LIN {X 0,Y 320.282,Z 387.307,A -85,B 0,C 180,E1 -15901.85,E2 -15901.85} C_VEL
LIN {X 0,Y 317.644,Z 401.035,A -85,B 0,C 180,E1 -15903.382,E2 -15903.382} C_VEL
LIN {X 0,Y 315.007,Z 413.467,A -85,B 0,C 180,E1 -15905.095,E2 -15905.095} C_VEL
LIN {X 0,Y 312.778,Z 423.901,A -85,B 0,C 180,E1 -15906.846,E2 -15906.846} C_VEL
LIN {X 0,Y 310.716,Z 433.586,A -85,B 0,C 180,E1 -15908.783,E2 -15908.783} C_VEL
LIN {X 0,Y 308.469,Z 443.101,A -85,B 0,C 180,E1 -15911.055,E2 -15911.055} C_VEL
LIN {X 0,Y 306.764,Z 451.036,A -85,B 0,C 180,E1 -15913.359,E2 -15913.359} C_VEL
LIN {X 0,Y 305.36,Z 458.451,A -85,B 0,C 180,E1 -15916.015,E2 -15916.015} C_VEL
LIN {X 0,Y 304.367,Z 464.336,A -85,B 0,C 180,E1 -15918.681,E2 -15918.681} C_VEL
LIN {X 0,Y 303.943,Z 467.84,A -85,B 0,C 180,E1 -15920.685,E2 -15920.685} C_VEL
LIN {X 0,Y 303.628,Z 471.382,A -85,B 0,C 180,E1 -15923.354,E2 -15923.354} C_VEL
LIN {X 0,Y 303.568,Z 473.714,A -85,B 0,C 180,E1 -15926.017,E2 -15926.017} C_VEL
LIN {X 0,Y 303.569,Z 474.886,A -85,B 0,C 180,E1 -15928.673,E2 -15928.673} C_VEL
LIN {X 0,Y 303.569,Z 474.883,A -85,B 0,C 180,E1 -15931.327,E2 -15931.327} C_VEL
LIN {X 0,Y 303.568,Z 473.697,A -85,B 0,C 180,E1 -15933.983,E2 -15933.983} C_VEL
LIN {X 0,Y 303.628,Z 471.354,A -85,B 0,C 180,E1 -15936.646,E2 -15936.646} C_VEL
LIN {X 0,Y 303.943,Z 467.807,A -85,B 0,C 180,E1 -15939.315,E2 -15939.315} C_VEL
LIN {X 0,Y 304.596,Z 462.968,A -85,B 0,C 180,E1 -15941.985,E2 -15941.985} C_VEL
LIN {X 0,Y 305.622,Z 456.707,A -85,B 0,C 180,E1 -15944.652,E2 -15944.652} C_VEL
LIN {X 0,Y 307.21,Z 448.855,A -85,B 0,C 180,E1 -15947.301,E2 -15947.301} C_VEL
LIN {X 0,Y 308.97,Z 440.507,A -85,B 0,C 180,E1 -15949.604,E2 -15949.604} C_VEL
LIN {X 0,Y 311.289,Z 430.696,A -85,B 0,C 180,E1 -15951.821,E2 -15951.821} C_VEL
LIN {X 0,Y 313.52,Z 420.19,A -85,B 0,C 180,E1 -15953.797,E2 -15953.797} C_VEL
LIN {X 0,Y 316.153,Z 407.953,A -85,B 0,C 180,E1 -15955.689,E2 -15955.689} C_VEL
LIN {X 0,Y 318.912,Z 394.331,A -85,B 0,C 180,E1 -15957.389,E2 -15957.389} C_VEL
LIN {X 0,Y 321.417,Z 380.677,A -85,B 0,C 180,E1 -15958.754,E2 -15958.754} C_VEL
LIN {X 0,Y 323.433,Z 367.3,A -85,B 0,C 180,E1 -15959.83,E2 -15959.83} C_VEL
LIN {X 0,Y 325.217,Z 353.283,A -85,B 0,C 180,E1 -15960.7,E2 -15960.7} C_VEL
LIN {X 0,Y 326.763,Z 337.925,A -85,B 0,C 180,E1 -15961.392,E2 -15961.392} C_VEL
LIN {X 0,Y 327.693,Z 323.115,A -85,B 0,C 180,E1 -15961.834,E2 -15961.834} C_VEL
LIN {X 0,Y 330.786,Z 234.22,A -85,B 0,C 180,E1 -15963.753,E2 -15963.753} C_VEL
LIN {X 0,Y 331.307,Z 215.247,A -85,B 0,C 180,E1 -15964.177,E2 -15964.177} C_VEL
LIN {X 0,Y 328.979,Z 201.739,A -85,B 0,C 180,E1 -15964.801,E2 -15964.801} C_VEL
LIN {X 0,Y 319.968,Z 182.03,A -85,B 0,C 180,E1 -15966.456,E2 -15966.456} C_VEL
LIN {X 0,Y 313.395,Z 169.255,A -85,B 0,C 180,E1 -15967.703,E2 -15967.703} C_VEL
LIN {X 0,Y 309.541,Z 161.949,A -85,B 0,C 180,E1 -15968.469,E2 -15968.469} C_VEL
LIN {X 0,Y 306.572,Z 151.906,A -85,B 0,C 180,E1 -15971.668,E2 -15971.668} C_VEL
LIN {X 0,Y 305.43,Z 148.062,A -85,B 0,C 180,E1 -15972.974,E2 -15972.974} C_VEL
LIN {X 0,Y 305.455,Z 148.059,A -85,B 0,C 180,E1 -15977.414,E2 -15977.414} C_VEL
LIN {X 0,Y 305.468,Z 148.053,A -85,B 0,C 180,E1 -15981.597,E2 -15981.597} C_VEL
LIN {X 0,Y 305.463,Z 148.054,A -85,B 0,C 180,E1 -15984.887,E2 -15984.887} C_VEL
LIN {X 0,Y 305.453,Z 148.058,A -85,B 0,C 180,E1 -15988.355,E2 -15988.355} C_VEL
LIN {X 0,Y 305.522,Z 148.05,A -85,B 0,C 180,E1 -15991.114,E2 -15991.114} C_VEL
LIN {X 0,Y 305.573,Z 148.045,A -85,B 0,C 180,E1 -15994.088,E2 -15994.088} C_VEL
LIN {X 0,Y 305.502,Z 148.056,A -85,B 0,C 180,E1 -15998.403,E2 -15998.403} C_VEL
LIN {X 0,Y 305.592,Z 148.044,A -85,B 0,C 180,E1 -16001.218,E2 -16001.218} C_VEL
LIN {X 0,Y 305.651,Z 148.037,A -85,B 0,C 180,E1 -16005.349,E2 -16005.349} C_VEL
LIN {X 0,Y 305.626,Z 148.04,A -85,B 0,C 180,E1 -16009.399,E2 -16009.399} C_VEL
LIN {X 0,Y 305.748,Z 148.015,A -85,B 0,C 180,E1 -16012.073,E2 -16012.073} C_VEL
LIN {X 0,Y 305.668,Z 148.031,A -85,B 0,C 180,E1 -16014.723,E2 -16014.723} C_VEL
LIN {X 0,Y 305.942,Z 147.999,A -85,B 0,C 180,E1 -16018.684,E2 -16018.684} C_VEL
LIN {X 0,Y 305.949,Z 147.996,A -85,B 0,C 180,E1 -16021.316,E2 -16021.316} C_VEL
LIN {X 0,Y 305.789,Z 148.021,A -85,B 0,C 180,E1 -16026.599,E2 -16026.599} C_VEL
LIN {X 0,Y 305.696,Z 148.022,A -85,B 0,C 180,E1 -16029.261,E2 -16029.261} C_VEL
LIN {X 0,Y 305.573,Z 148.037,A -85,B 0,C 180,E1 -16033.297,E2 -16033.297} C_VEL
LIN {X 0,Y 305.533,Z 148.043,A -85,B 0,C 180,E1 -16037.4,E2 -16037.4} C_VEL
LIN {X 0,Y 305.501,Z 148.051,A -85,B 0,C 180,E1 -16040.186,E2 -16040.186} C_VEL
LIN {X 0,Y 305.475,Z 148.051,A -85,B 0,C 180,E1 -16044.464,E2 -16044.464} C_VEL
LIN {X 0,Y 305.455,Z 148.035,A -85,B 0,C 180,E1 -16047.398,E2 -16047.398} C_VEL
LIN {X 0,Y 305.431,Z 148.063,A -85,B 0,C 180,E1 -16050.413,E2 -16050.413} C_VEL
LIN {X 0,Y 305.466,Z 148.053,A -85,B 0,C 180,E1 -16054.078,E2 -16054.078} C_VEL
LIN {X 0,Y 305.455,Z 148.057,A -85,B 0,C 180,E1 -16056.742,E2 -16056.742} C_VEL
LIN {X 0,Y 305.41,Z 148.062,A -85,B 0,C 180,E1 -16060.59,E2 -16060.59} C_VEL
LIN {X 0,Y 305.421,Z 148.064,A -85,B 0,C 180,E1 -16063.656,E2 -16063.656} C_VEL
LIN {X 0,Y 305.436,Z 148.064,A -85,B 0,C 180,E1 -16067.418,E2 -16067.418} C_VEL
LIN {X 0,Y 305.445,Z 148.217,A -85,B 0,C 180,E1 -16070.766,E2 -16070.766} C_VEL
LIN {X 0,Y 305.708,Z 149.306,A -85,B 0,C 180,E1 -16071.033,E2 -16071.033} C_VEL
LIN {X 0,Y 307.015,Z 151.728,A -85,B 0,C 180,E1 -16071.303,E2 -16071.303} C_VEL
LIN {X 0,Y 311.31,Z 158.512,A -85,B 0,C 180,E1 -16072.134,E2 -16072.134} C_VEL
LIN {X 0,Y 319.576,Z 173.575,A -85,B 0,C 180,E1 -16073.7,E2 -16073.7} C_VEL
LIN {X 0,Y 326.924,Z 188.491,A -85,B 0,C 180,E1 -16075.041,E2 -16075.041} C_VEL
LIN {X 0,Y 331.801,Z 199.525,A -85,B 0,C 180,E1 -16075.917,E2 -16075.917} C_VEL
LIN {X 0,Y 330.462,Z 240.875,A -85,B 0,C 180,E1 -16076.819,E2 -16076.819} C_VEL
LIN {X 0,Y 327.848,Z 313.454,A -85,B 0,C 180,E1 -16078.408,E2 -16078.408} C_VEL
LIN {X 0,Y 326.848,Z 327.773,A -85,B 0,C 180,E1 -16078.932,E2 -16078.932} C_VEL
LIN {X 0,Y 325.558,Z 340.971,A -85,B 0,C 180,E1 -16079.614,E2 -16079.614} C_VEL
LIN {X 0,Y 323.859,Z 355.279,A -85,B 0,C 180,E1 -16080.595,E2 -16080.595} C_VEL
LIN {X 0,Y 321.646,Z 369.25,A -85,B 0,C 180,E1 -16081.803,E2 -16081.803} C_VEL
LIN {X 0,Y 319.391,Z 382.018,A -85,B 0,C 180,E1 -16083.186,E2 -16083.186} C_VEL
LIN {X 0,Y 316.811,Z 394.879,A -85,B 0,C 180,E1 -16084.896,E2 -16084.896} C_VEL
LIN {X 0,Y 314.858,Z 403.853,A -85,B 0,C 180,E1 -16086.31,E2 -16086.31} C_VEL
LIN {X 0,Y 312.98,Z 412.416,A -85,B 0,C 180,E1 -16087.906,E2 -16087.906} C_VEL
LIN {X 0,Y 310.65,Z 422.648,A -85,B 0,C 180,E1 -16090.162,E2 -16090.162} C_VEL
LIN {X 0,Y 308.592,Z 431.143,A -85,B 0,C 180,E1 -16092.437,E2 -16092.437} C_VEL
LIN {X 0,Y 307.076,Z 438.205,A -85,B 0,C 180,E1 -16094.74,E2 -16094.74} C_VEL
LIN {X 0,Y 305.643,Z 444.756,A -85,B 0,C 180,E1 -16097.382,E2 -16097.382} C_VEL
LIN {X 0,Y 304.74,Z 449.87,A -85,B 0,C 180,E1 -16100.04,E2 -16100.04} C_VEL
LIN {X 0,Y 304.281,Z 452.816,A -85,B 0,C 180,E1 -16102.034,E2 -16102.034} C_VEL
LIN {X 0,Y 303.871,Z 455.7,A -85,B 0,C 180,E1 -16104.692,E2 -16104.692} C_VEL
LIN {X 0,Y 303.673,Z 457.433,A -85,B 0,C 180,E1 -16107.347,E2 -16107.347} C_VEL
LIN {X 0,Y 303.609,Z 458.038,A -85,B 0,C 180,E1 -16110,E2 -16110} C_VEL
LIN {X 0,Y 303.672,Z 457.475,A -85,B 0,C 180,E1 -16112.653,E2 -16112.653} C_VEL
LIN {X 0,Y 303.87,Z 455.798,A -85,B 0,C 180,E1 -16115.308,E2 -16115.308} C_VEL
LIN {X 0,Y 304.274,Z 452.967,A -85,B 0,C 180,E1 -16117.966,E2 -16117.966} C_VEL
LIN {X 0,Y 304.917,Z 448.913,A -85,B 0,C 180,E1 -16120.626,E2 -16120.626} C_VEL
LIN {X 0,Y 305.957,Z 443.534,A -85,B 0,C 180,E1 -16123.28,E2 -16123.28} C_VEL
LIN {X 0,Y 307.039,Z 438.509,A -85,B 0,C 180,E1 -16125.262,E2 -16125.262} C_VEL
LIN {X 0,Y 308.808,Z 430.409,A -85,B 0,C 180,E1 -16127.893,E2 -16127.893} C_VEL
LIN {X 0,Y 310.834,Z 421.751,A -85,B 0,C 180,E1 -16130.17,E2 -16130.17} C_VEL
LIN {X 0,Y 313.314,Z 411.331,A -85,B 0,C 180,E1 -16132.416,E2 -16132.416} C_VEL
LIN {X 0,Y 315.625,Z 400.631,A -85,B 0,C 180,E1 -16134.326,E2 -16134.326} C_VEL
LIN {X 0,Y 317.873,Z 390.102,A -85,B 0,C 180,E1 -16135.891,E2 -16135.891} C_VEL
LIN {X 0,Y 320.214,Z 377.582,A -85,B 0,C 180,E1 -16137.446,E2 -16137.446} C_VEL
LIN {X 0,Y 322.645,Z 363.942,A -85,B 0,C 180,E1 -16138.799,E2 -16138.799} C_VEL
LIN {X 0,Y 324.486,Z 350.567,A -85,B 0,C 180,E1 -16139.878,E2 -16139.878} C_VEL
LIN {X 0,Y 326.118,Z 335.98,A -85,B 0,C 180,E1 -16140.785,E2 -16140.785} C_VEL
LIN {X 0,Y 327.451,Z 320.953,A -85,B 0,C 180,E1 -16141.454,E2 -16141.454} C_VEL
LIN {X 0,Y 328.374,Z 305.322,A -85,B 0,C 180,E1 -16141.896,E2 -16141.896} C_VEL
LIN {X 0,Y 331.426,Z 216.152,A -85,B 0,C 180,E1 -16143.819,E2 -16143.819} C_VEL
LIN {X 0,Y 331.182,Z 212.313,A -85,B 0,C 180,E1 -16143.946,E2 -16143.946} C_VEL
LIN {X 0,Y 329.668,Z 206.897,A -85,B 0,C 180,E1 -16144.265,E2 -16144.265} C_VEL
LIN {X 0,Y 327.311,Z 201.936,A -85,B 0,C 180,E1 -16144.678,E2 -16144.678} C_VEL
LIN {X 0,Y 321.759,Z 192.218,A -85,B 0,C 180,E1 -16145.631,E2 -16145.631} C_VEL
LIN {X 0,Y 320.189,Z 188.776,A -85,B 0,C 180,E1 -16145.927,E2 -16145.927} C_VEL
LIN {X 0,Y 311.448,Z 171.517,A -85,B 0,C 180,E1 -16147.6,E2 -16147.6} C_VEL
LIN {X 0,Y 304.534,Z 159.472,A -85,B 0,C 180,E1 -16148.973,E2 -16148.973} C_VEL
LIN {X 0,Y 300.514,Z 153.176,A -85,B 0,C 180,E1 -16149.792,E2 -16149.792} C_VEL
LIN {X 0,Y 298.852,Z 150.776,A -85,B 0,C 180,E1 -16150.134,E2 -16150.134} C_VEL
LIN {X 0,Y 298.381,Z 148.995,A -85,B 0,C 180,E1 -16150.317,E2 -16150.317} C_VEL
LIN {X 0,Y 298.371,Z 148.945,A -85,B 0,C 180,E1 -16153.097,E2 -16153.097} C_VEL
LIN {X 0,Y 298.37,Z 148.928,A -85,B 0,C 180,E1 -16156.915,E2 -16156.915} C_VEL
LIN {X 0,Y 298.357,Z 148.938,A -85,B 0,C 180,E1 -16161.018,E2 -16161.018} C_VEL
LIN {X 0,Y 298.405,Z 148.924,A -85,B 0,C 180,E1 -16163.928,E2 -16163.928} C_VEL
LIN {X 0,Y 298.393,Z 148.925,A -85,B 0,C 180,E1 -16167.199,E2 -16167.199} C_VEL
LIN {X 0,Y 298.405,Z 148.939,A -85,B 0,C 180,E1 -16171.898,E2 -16171.898} C_VEL
LIN {X 0,Y 298.422,Z 148.935,A -85,B 0,C 180,E1 -16174.918,E2 -16174.918} C_VEL
LIN {X 0,Y 298.417,Z 148.937,A -85,B 0,C 180,E1 -16179.313,E2 -16179.313} C_VEL
LIN {X 0,Y 298.452,Z 148.925,A -85,B 0,C 180,E1 -16182.174,E2 -16182.174} C_VEL
LIN {X 0,Y 298.588,Z 148.914,A -85,B 0,C 180,E1 -16184.994,E2 -16184.994} C_VEL
LIN {X 0,Y 298.586,Z 148.916,A -85,B 0,C 180,E1 -16189.146,E2 -16189.146} C_VEL
LIN {X 0,Y 298.699,Z 148.896,A -85,B 0,C 180,E1 -16191.884,E2 -16191.884} C_VEL
LIN {X 0,Y 298.629,Z 148.904,A -85,B 0,C 180,E1 -16194.598,E2 -16194.598} C_VEL
LIN {X 0,Y 298.914,Z 148.873,A -85,B 0,C 180,E1 -16198.653,E2 -16198.653} C_VEL
LIN {X 0,Y 298.911,Z 148.871,A -85,B 0,C 180,E1 -16201.347,E2 -16201.347} C_VEL
LIN {X 0,Y 298.637,Z 148.901,A -85,B 0,C 180,E1 -16205.401,E2 -16205.401} C_VEL
LIN {X 0,Y 298.71,Z 148.894,A -85,B 0,C 180,E1 -16208.82,E2 -16208.82} C_VEL
LIN {X 0,Y 298.553,Z 148.921,A -85,B 0,C 180,E1 -16212.231,E2 -16212.231} C_VEL
LIN {X 0,Y 298.55,Z 148.92,A -85,B 0,C 180,E1 -16215.168,E2 -16215.168} C_VEL
LIN {X 0,Y 298.51,Z 148.923,A -85,B 0,C 180,E1 -16219.245,E2 -16219.245} C_VEL
LIN {X 0,Y 298.426,Z 148.937,A -85,B 0,C 180,E1 -16223.6,E2 -16223.6} C_VEL
LIN {X 0,Y 298.418,Z 148.93,A -85,B 0,C 180,E1 -16226.581,E2 -16226.581} C_VEL
LIN {X 0,Y 298.402,Z 148.94,A -85,B 0,C 180,E1 -16229.643,E2 -16229.643} C_VEL
LIN {X 0,Y 298.394,Z 148.936,A -85,B 0,C 180,E1 -16232.8,E2 -16232.8} C_VEL
LIN {X 0,Y 298.447,Z 148.927,A -85,B 0,C 180,E1 -16236.807,E2 -16236.807} C_VEL
LIN {X 0,Y 298.389,Z 148.943,A -85,B 0,C 180,E1 -16241.088,E2 -16241.088} C_VEL
LIN {X 0,Y 298.399,Z 148.938,A -85,B 0,C 180,E1 -16243.103,E2 -16243.103} C_VEL
LIN {X 0,Y 298.387,Z 149.027,A -85,B 0,C 180,E1 -16246.102,E2 -16246.102} C_VEL
LIN {X 0,Y 301.743,Z 159.889,A -85,B 0,C 180,E1 -16249.803,E2 -16249.803} C_VEL
LIN {X 0,Y 302.402,Z 162.037,A -85,B 0,C 180,E1 -16250.425,E2 -16250.425} C_VEL
LIN {X 0,Y 312.165,Z 180.214,A -85,B 0,C 180,E1 -16252.4,E2 -16252.4} C_VEL
LIN {X 0,Y 320.694,Z 198.338,A -85,B 0,C 180,E1 -16254.049,E2 -16254.049} C_VEL
LIN {X 0,Y 323.674,Z 205.479,A -85,B 0,C 180,E1 -16254.618,E2 -16254.618} C_VEL
LIN {X 0,Y 325.588,Z 217.919,A -85,B 0,C 180,E1 -16255.183,E2 -16255.183} C_VEL
LIN {X 0,Y 321.554,Z 326.838,A -85,B 0,C 180,E1 -16257.577,E2 -16257.577} C_VEL
LIN {X 0,Y 320.415,Z 341.93,A -85,B 0,C 180,E1 -16258.097,E2 -16258.097} C_VEL
LIN {X 0,Y 318.626,Z 357.365,A -85,B 0,C 180,E1 -16258.871,E2 -16258.871} C_VEL
LIN {X 0,Y 316.699,Z 371.078,A -85,B 0,C 180,E1 -16259.81,E2 -16259.81} C_VEL
LIN {X 0,Y 314.58,Z 383.941,A -85,B 0,C 180,E1 -16260.927,E2 -16260.927} C_VEL
LIN {X 0,Y 312.061,Z 396.955,A -85,B 0,C 180,E1 -16262.322,E2 -16262.322} C_VEL
LIN {X 0,Y 309.265,Z 410.05,A -85,B 0,C 180,E1 -16264.058,E2 -16264.058} C_VEL
LIN {X 0,Y 306.578,Z 421.907,A -85,B 0,C 180,E1 -16265.989,E2 -16265.989} C_VEL
LIN {X 0,Y 304.366,Z 432.073,A -85,B 0,C 180,E1 -16268.004,E2 -16268.004} C_VEL
LIN {X 0,Y 301.959,Z 441.661,A -85,B 0,C 180,E1 -16270.276,E2 -16270.276} C_VEL
LIN {X 0,Y 300.111,Z 449.82,A -85,B 0,C 180,E1 -16272.628,E2 -16272.628} C_VEL
LIN {X 0,Y 298.712,Z 456.572,A -85,B 0,C 180,E1 -16275.001,E2 -16275.001} C_VEL
LIN {X 0,Y 297.615,Z 462.812,A -85,B 0,C 180,E1 -16277.729,E2 -16277.729} C_VEL
LIN {X 0,Y 296.896,Z 467.641,A -85,B 0,C 180,E1 -16280.462,E2 -16280.462} C_VEL
LIN {X 0,Y 296.548,Z 471.183,A -85,B 0,C 180,E1 -16283.195,E2 -16283.195} C_VEL
LIN {X 0,Y 296.469,Z 473.515,A -85,B 0,C 180,E1 -16285.922,E2 -16285.922} C_VEL
LIN {X 0,Y 296.488,Z 474.688,A -85,B 0,C 180,E1 -16288.642,E2 -16288.642} C_VEL
LIN {X 0,Y 296.488,Z 474.684,A -85,B 0,C 180,E1 -16291.358,E2 -16291.358} C_VEL
LIN {X 0,Y 296.469,Z 473.498,A -85,B 0,C 180,E1 -16294.078,E2 -16294.078} C_VEL
LIN {X 0,Y 296.547,Z 471.154,A -85,B 0,C 180,E1 -16296.805,E2 -16296.805} C_VEL
LIN {X 0,Y 296.895,Z 467.606,A -85,B 0,C 180,E1 -16299.538,E2 -16299.538} C_VEL
LIN {X 0,Y 297.609,Z 462.767,A -85,B 0,C 180,E1 -16302.271,E2 -16302.271} C_VEL
LIN {X 0,Y 298.657,Z 456.504,A -85,B 0,C 180,E1 -16305.002,E2 -16305.002} C_VEL
LIN {X 0,Y 300.353,Z 448.652,A -85,B 0,C 180,E1 -16307.709,E2 -16307.709} C_VEL
LIN {X 0,Y 302.223,Z 440.305,A -85,B 0,C 180,E1 -16310.06,E2 -16310.06} C_VEL
LIN {X 0,Y 304.537,Z 430.85,A -85,B 0,C 180,E1 -16312.248,E2 -16312.248} C_VEL
LIN {X 0,Y 306.991,Z 419.987,A -85,B 0,C 180,E1 -16314.335,E2 -16314.335} C_VEL
LIN {X 0,Y 309.728,Z 407.75,A -85,B 0,C 180,E1 -16316.262,E2 -16316.262} C_VEL
LIN {X 0,Y 312.58,Z 394.127,A -85,B 0,C 180,E1 -16317.992,E2 -16317.992} C_VEL
LIN {X 0,Y 315.185,Z 380.472,A -85,B 0,C 180,E1 -16319.377,E2 -16319.377} C_VEL
LIN {X 0,Y 317.382,Z 366.271,A -85,B 0,C 180,E1 -16320.53,E2 -16320.53} C_VEL
LIN {X 0,Y 319.32,Z 351.754,A -85,B 0,C 180,E1 -16321.423,E2 -16321.423} C_VEL
LIN {X 0,Y 320.806,Z 336.793,A -85,B 0,C 180,E1 -16322.09,E2 -16322.09} C_VEL
LIN {X 0,Y 321.751,Z 321.39,A -85,B 0,C 180,E1 -16322.54,E2 -16322.54} C_VEL
LIN {X 0,Y 324.847,Z 235.601,A -85,B 0,C 180,E1 -16324.414,E2 -16324.414} C_VEL
LIN {X 0,Y 325.425,Z 216.339,A -85,B 0,C 180,E1 -16324.849,E2 -16324.849} C_VEL
LIN {X 0,Y 323.337,Z 204.486,A -85,B 0,C 180,E1 -16325.42,E2 -16325.42} C_VEL
LIN {X 0,Y 314.903,Z 185.886,A -85,B 0,C 180,E1 -16327.027,E2 -16327.027} C_VEL
LIN {X 0,Y 308.532,Z 173.387,A -85,B 0,C 180,E1 -16328.279,E2 -16328.279} C_VEL
LIN {X 0,Y 303.597,Z 164.547,A -85,B 0,C 180,E1 -16329.275,E2 -16329.275} C_VEL
LIN {X 0,Y 302.195,Z 161.662,A -85,B 0,C 180,E1 -16329.591,E2 -16329.591} C_VEL
LIN {X 0,Y 299.183,Z 151.637,A -85,B 0,C 180,E1 -16332.94,E2 -16332.94} C_VEL
LIN {X 0,Y 298.385,Z 148.942,A -85,B 0,C 180,E1 -16333.954,E2 -16333.954} C_VEL
LIN {X 0,Y 298.403,Z 148.935,A -85,B 0,C 180,E1 -16336.921,E2 -16336.921} C_VEL
LIN {X 0,Y 298.399,Z 148.935,A -85,B 0,C 180,E1 -16341.008,E2 -16341.008} C_VEL
LIN {X 0,Y 298.418,Z 148.929,A -85,B 0,C 180,E1 -16343.93,E2 -16343.93} C_VEL
LIN {X 0,Y 298.397,Z 148.938,A -85,B 0,C 180,E1 -16347.983,E2 -16347.983} C_VEL
LIN {X 0,Y 298.465,Z 148.93,A -85,B 0,C 180,E1 -16351.905,E2 -16351.905} C_VEL
LIN {X 0,Y 298.487,Z 148.931,A -85,B 0,C 180,E1 -16354.924,E2 -16354.924} C_VEL
LIN {X 0,Y 298.451,Z 148.927,A -85,B 0,C 180,E1 -16359.316,E2 -16359.316} C_VEL
LIN {X 0,Y 298.54,Z 148.923,A -85,B 0,C 180,E1 -16362.18,E2 -16362.18} C_VEL
LIN {X 0,Y 298.595,Z 148.915,A -85,B 0,C 180,E1 -16364.995,E2 -16364.995} C_VEL
LIN {X 0,Y 298.585,Z 148.918,A -85,B 0,C 180,E1 -16369.146,E2 -16369.146} C_VEL
LIN {X 0,Y 298.7,Z 148.892,A -85,B 0,C 180,E1 -16371.884,E2 -16371.884} C_VEL
LIN {X 0,Y 298.637,Z 148.908,A -85,B 0,C 180,E1 -16374.599,E2 -16374.599} C_VEL
LIN {X 0,Y 298.91,Z 148.875,A -85,B 0,C 180,E1 -16378.653,E2 -16378.653} C_VEL
LIN {X 0,Y 298.915,Z 148.873,A -85,B 0,C 180,E1 -16381.347,E2 -16381.347} C_VEL
LIN {X 0,Y 298.737,Z 148.898,A -85,B 0,C 180,E1 -16386.755,E2 -16386.755} C_VEL
LIN {X 0,Y 298.627,Z 148.903,A -85,B 0,C 180,E1 -16389.482,E2 -16389.482} C_VEL
LIN {X 0,Y 298.525,Z 148.915,A -85,B 0,C 180,E1 -16393.617,E2 -16393.617} C_VEL
LIN {X 0,Y 298.464,Z 148.926,A -85,B 0,C 180,E1 -16396.414,E2 -16396.414} C_VEL
LIN {X 0,Y 298.488,Z 148.93,A -85,B 0,C 180,E1 -16399.641,E2 -16399.641} C_VEL
LIN {X 0,Y 298.422,Z 148.936,A -85,B 0,C 180,E1 -16403.601,E2 -16403.601} C_VEL
LIN {X 0,Y 298.408,Z 148.908,A -85,B 0,C 180,E1 -16406.582,E2 -16406.582} C_VEL
LIN {X 0,Y 298.394,Z 148.943,A -85,B 0,C 180,E1 -16409.644,E2 -16409.644} C_VEL
LIN {X 0,Y 298.394,Z 148.941,A -85,B 0,C 180,E1 -16412.801,E2 -16412.801} C_VEL
LIN {X 0,Y 298.429,Z 148.931,A -85,B 0,C 180,E1 -16416.803,E2 -16416.803} C_VEL
LIN {X 0,Y 298.375,Z 148.937,A -85,B 0,C 180,E1 -16419.492,E2 -16419.492} C_VEL
LIN {X 0,Y 298.371,Z 148.94,A -85,B 0,C 180,E1 -16423.097,E2 -16423.097} C_VEL
LIN {X 0,Y 298.371,Z 148.941,A -85,B 0,C 180,E1 -16426.915,E2 -16426.915} C_VEL
LIN {X 0,Y 298.384,Z 149.054,A -85,B 0,C 180,E1 -16429.835,E2 -16429.835} C_VEL
LIN {X 0,Y 299.497,Z 151.955,A -85,B 0,C 180,E1 -16430.139,E2 -16430.139} C_VEL
LIN {X 0,Y 301.215,Z 154.199,A -85,B 0,C 180,E1 -16430.482,E2 -16430.482} C_VEL
LIN {X 0,Y 308.565,Z 166.283,A -85,B 0,C 180,E1 -16431.959,E2 -16431.959} C_VEL
LIN {X 0,Y 316.644,Z 181.593,A -85,B 0,C 180,E1 -16433.528,E2 -16433.528} C_VEL
LIN {X 0,Y 324.076,Z 197.348,A -85,B 0,C 180,E1 -16434.922,E2 -16434.922} C_VEL
LIN {X 0,Y 325.912,Z 201.621,A -85,B 0,C 180,E1 -16435.262,E2 -16435.262} C_VEL
LIN {X 0,Y 323.491,Z 271.441,A -85,B 0,C 180,E1 -16436.801,E2 -16436.801} C_VEL
LIN {X 0,Y 321.834,Z 313.669,A -85,B 0,C 180,E1 -16437.748,E2 -16437.748} C_VEL
LIN {X 0,Y 320.791,Z 327.984,A -85,B 0,C 180,E1 -16438.278,E2 -16438.278} C_VEL
LIN {X 0,Y 319.385,Z 341.953,A -85,B 0,C 180,E1 -16439.018,E2 -16439.018} C_VEL
LIN {X 0,Y 317.695,Z 355.485,A -85,B 0,C 180,E1 -16439.966,E2 -16439.966} C_VEL
LIN {X 0,Y 315.416,Z 369.454,A -85,B 0,C 180,E1 -16441.194,E2 -16441.194} C_VEL
LIN {X 0,Y 313.071,Z 382.221,A -85,B 0,C 180,E1 -16442.6,E2 -16442.6} C_VEL
LIN {X 0,Y 310.37,Z 395.083,A -85,B 0,C 180,E1 -16444.338,E2 -16444.338} C_VEL
LIN {X 0,Y 308.06,Z 405.449,A -85,B 0,C 180,E1 -16446.036,E2 -16446.036} C_VEL
LIN {X 0,Y 306.021,Z 414.236,A -85,B 0,C 180,E1 -16447.732,E2 -16447.732} C_VEL
LIN {X 0,Y 303.622,Z 424.194,A -85,B 0,C 180,E1 -16450.036,E2 -16450.036} C_VEL
LIN {X 0,Y 301.511,Z 432.453,A -85,B 0,C 180,E1 -16452.361,E2 -16452.361} C_VEL
LIN {X 0,Y 299.83,Z 440.199,A -85,B 0,C 180,E1 -16455.058,E2 -16455.058} C_VEL
LIN {X 0,Y 298.391,Z 446.367,A -85,B 0,C 180,E1 -16457.762,E2 -16457.762} C_VEL
LIN {X 0,Y 297.538,Z 451.123,A -85,B 0,C 180,E1 -16460.483,E2 -16460.483} C_VEL
LIN {X 0,Y 297,Z 454.604,A -85,B 0,C 180,E1 -16463.205,E2 -16463.205} C_VEL
LIN {X 0,Y 296.703,Z 456.905,A -85,B 0,C 180,E1 -16465.925,E2 -16465.925} C_VEL
LIN {X 0,Y 296.526,Z 458.08,A -85,B 0,C 180,E1 -16468.642,E2 -16468.642} C_VEL
LIN {X 0,Y 296.526,Z 458.094,A -85,B 0,C 180,E1 -16471.358,E2 -16471.358} C_VEL
LIN {X 0,Y 296.703,Z 456.975,A -85,B 0,C 180,E1 -16474.075,E2 -16474.075} C_VEL
LIN {X 0,Y 296.999,Z 454.729,A -85,B 0,C 180,E1 -16476.795,E2 -16476.795} C_VEL
LIN {X 0,Y 297.518,Z 451.297,A -85,B 0,C 180,E1 -16479.518,E2 -16479.518} C_VEL
LIN {X 0,Y 298.361,Z 446.597,A -85,B 0,C 180,E1 -16482.24,E2 -16482.24} C_VEL
LIN {X 0,Y 299.801,Z 440.499,A -85,B 0,C 180,E1 -16484.944,E2 -16484.944} C_VEL
LIN {X 0,Y 301.48,Z 432.824,A -85,B 0,C 180,E1 -16487.641,E2 -16487.641} C_VEL
LIN {X 0,Y 303.501,Z 424.632,A -85,B 0,C 180,E1 -16489.972,E2 -16489.972} C_VEL
LIN {X 0,Y 305.945,Z 414.758,A -85,B 0,C 180,E1 -16492.274,E2 -16492.274} C_VEL
LIN {X 0,Y 308.306,Z 404.555,A -85,B 0,C 180,E1 -16494.241,E2 -16494.241} C_VEL
LIN {X 0,Y 310.981,Z 392.574,A -85,B 0,C 180,E1 -16496.148,E2 -16496.148} C_VEL
LIN {X 0,Y 313.414,Z 380.478,A -85,B 0,C 180,E1 -16497.73,E2 -16497.73} C_VEL
LIN {X 0,Y 315.879,Z 367.325,A -85,B 0,C 180,E1 -16499.124,E2 -16499.124} C_VEL
LIN {X 0,Y 318.067,Z 352.667,A -85,B 0,C 180,E1 -16500.374,E2 -16500.374} C_VEL
LIN {X 0,Y 319.852,Z 338.161,A -85,B 0,C 180,E1 -16501.318,E2 -16501.318} C_VEL
LIN {X 0,Y 321.25,Z 323.005,A -85,B 0,C 180,E1 -16502.041,E2 -16502.041} C_VEL
LIN {X 0,Y 322.237,Z 307.077,A -85,B 0,C 180,E1 -16502.531,E2 -16502.531} C_VEL
LIN {X 0,Y 326.093,Z 201.988,A -85,B 0,C 180,E1 -16504.826,E2 -16504.826} C_VEL
LIN {X 0,Y 320.189,Z 188.776,A -85,B 0,C 180,E1 -16505.927,E2 -16505.927} C_VEL
LIN {X 0,Y 317.58,Z 184.209,A -85,B 0,C 180,E1 -16506.397,E2 -16506.397} C_VEL
LIN {X 0,Y 314.188,Z 180.465,A -85,B 0,C 180,E1 -16506.963,E2 -16506.963} C_VEL
LIN {X 0,Y 305.628,Z 172.6,A -85,B 0,C 180,E1 -16508.419,E2 -16508.419} C_VEL
LIN {X 0,Y 302.592,Z 168.468,A -85,B 0,C 180,E1 -16509.003,E2 -16509.003} C_VEL
LIN {X 0,Y 297.933,Z 160.898,A -85,B 0,C 180,E1 -16509.971,E2 -16509.971} C_VEL
LIN {X 0,Y 295.918,Z 157.822,A -85,B 0,C 180,E1 -16510.397,E2 -16510.397} C_VEL
LIN {X 0,Y 293.645,Z 154.259,A -85,B 0,C 180,E1 -16510.891,E2 -16510.891} C_VEL
LIN {X 0,Y 291.806,Z 151.71,A -85,B 0,C 180,E1 -16511.288,E2 -16511.288} C_VEL
LIN {X 0,Y 291.304,Z 149.828,A -85,B 0,C 180,E1 -16511.461,E2 -16511.461} C_VEL
LIN {X 0,Y 291.283,Z 149.827,A -85,B 0,C 180,E1 -16515.597,E2 -16515.597} C_VEL
LIN {X 0,Y 291.295,Z 149.821,A -85,B 0,C 180,E1 -16519.351,E2 -16519.351} C_VEL
LIN {X 0,Y 291.388,Z 149.789,A -85,B 0,C 180,E1 -16522.916,E2 -16522.916} C_VEL
LIN {X 0,Y 291.345,Z 149.815,A -85,B 0,C 180,E1 -16526.301,E2 -16526.301} C_VEL
LIN {X 0,Y 291.339,Z 149.801,A -85,B 0,C 180,E1 -16530.277,E2 -16530.277} C_VEL
LIN {X 0,Y 291.347,Z 149.811,A -85,B 0,C 180,E1 -16534.265,E2 -16534.265} C_VEL
LIN {X 0,Y 291.351,Z 149.811,A -85,B 0,C 180,E1 -16537.297,E2 -16537.297} C_VEL
LIN {X 0,Y 291.387,Z 149.813,A -85,B 0,C 180,E1 -16540.265,E2 -16540.265} C_VEL
LIN {X 0,Y 291.482,Z 149.8,A -85,B 0,C 180,E1 -16544.678,E2 -16544.678} C_VEL
LIN {X 0,Y 291.531,Z 149.795,A -85,B 0,C 180,E1 -16548.88,E2 -16548.88} C_VEL
LIN {X 0,Y 291.653,Z 149.772,A -85,B 0,C 180,E1 -16551.687,E2 -16551.687} C_VEL
LIN {X 0,Y 291.599,Z 149.78,A -85,B 0,C 180,E1 -16554.468,E2 -16554.468} C_VEL
LIN {X 0,Y 291.881,Z 149.75,A -85,B 0,C 180,E1 -16558.62,E2 -16558.62} C_VEL
LIN {X 0,Y 291.878,Z 149.747,A -85,B 0,C 180,E1 -16561.38,E2 -16561.38} C_VEL
LIN {X 0,Y 291.606,Z 149.778,A -85,B 0,C 180,E1 -16565.532,E2 -16565.532} C_VEL
LIN {X 0,Y 291.669,Z 149.77,A -85,B 0,C 180,E1 -16568.91,E2 -16568.91} C_VEL
LIN {X 0,Y 291.519,Z 149.797,A -85,B 0,C 180,E1 -16572.531,E2 -16572.531} C_VEL
LIN {X 0,Y 291.509,Z 149.799,A -85,B 0,C 180,E1 -16575.379,E2 -16575.379} C_VEL
LIN {X 0,Y 291.425,Z 149.811,A -85,B 0,C 180,E1 -16579.86,E2 -16579.86} C_VEL
LIN {X 0,Y 291.369,Z 149.818,A -85,B 0,C 180,E1 -16584.208,E2 -16584.208} C_VEL
LIN {X 0,Y 291.363,Z 149.813,A -85,B 0,C 180,E1 -16587.277,E2 -16587.277} C_VEL
LIN {X 0,Y 291.323,Z 149.824,A -85,B 0,C 180,E1 -16590.438,E2 -16590.438} C_VEL
LIN {X 0,Y 291.345,Z 149.809,A -85,B 0,C 180,E1 -16593.698,E2 -16593.698} C_VEL
LIN {X 0,Y 291.377,Z 149.808,A -85,B 0,C 180,E1 -16597.254,E2 -16597.254} C_VEL
LIN {X 0,Y 291.334,Z 149.817,A -85,B 0,C 180,E1 -16600.642,E2 -16600.642} C_VEL
LIN {X 0,Y 291.318,Z 149.818,A -85,B 0,C 180,E1 -16604.91,E2 -16604.91} C_VEL
LIN {X 0,Y 291.327,Z 149.827,A -85,B 0,C 180,E1 -16605.081,E2 -16605.081} C_VEL
LIN {X 0,Y 294.981,Z 161.592,A -85,B 0,C 180,E1 -16609.217,E2 -16609.217} C_VEL
LIN {X 0,Y 303.922,Z 177.912,A -85,B 0,C 180,E1 -16611.133,E2 -16611.133} C_VEL
LIN {X 0,Y 310.773,Z 191.526,A -85,B 0,C 180,E1 -16612.526,E2 -16612.526} C_VEL
LIN {X 0,Y 318.084,Z 208.052,A -85,B 0,C 180,E1 -16613.975,E2 -16613.975} C_VEL
LIN {X 0,Y 319.739,Z 218.75,A -85,B 0,C 180,E1 -16614.478,E2 -16614.478} C_VEL
LIN {X 0,Y 315.671,Z 325.152,A -85,B 0,C 180,E1 -16616.848,E2 -16616.848} C_VEL
LIN {X 0,Y 314.481,Z 340.825,A -85,B 0,C 180,E1 -16617.374,E2 -16617.374} C_VEL
LIN {X 0,Y 312.745,Z 355.871,A -85,B 0,C 180,E1 -16618.123,E2 -16618.123} C_VEL
LIN {X 0,Y 310.793,Z 369.4,A -85,B 0,C 180,E1 -16619.033,E2 -16619.033} C_VEL
LIN {X 0,Y 308.375,Z 383.747,A -85,B 0,C 180,E1 -16620.284,E2 -16620.284} C_VEL
LIN {X 0,Y 305.753,Z 396.758,A -85,B 0,C 180,E1 -16621.7,E2 -16621.7} C_VEL
LIN {X 0,Y 303.106,Z 408.779,A -85,B 0,C 180,E1 -16623.305,E2 -16623.305} C_VEL
LIN {X 0,Y 300.479,Z 419.917,A -85,B 0,C 180,E1 -16625.102,E2 -16625.102} C_VEL
LIN {X 0,Y 297.928,Z 430.876,A -85,B 0,C 180,E1 -16627.259,E2 -16627.259} C_VEL
LIN {X 0,Y 295.572,Z 440.204,A -85,B 0,C 180,E1 -16629.469,E2 -16629.469} C_VEL
LIN {X 0,Y 293.523,Z 448.537,A -85,B 0,C 180,E1 -16631.864,E2 -16631.864} C_VEL
LIN {X 0,Y 291.803,Z 456.372,A -85,B 0,C 180,E1 -16634.637,E2 -16634.637} C_VEL
LIN {X 0,Y 290.607,Z 462.612,A -85,B 0,C 180,E1 -16637.429,E2 -16637.429} C_VEL
LIN {X 0,Y 289.823,Z 467.441,A -85,B 0,C 180,E1 -16640.227,E2 -16640.227} C_VEL
LIN {X 0,Y 289.464,Z 470.983,A -85,B 0,C 180,E1 -16643.027,E2 -16643.027} C_VEL
LIN {X 0,Y 289.374,Z 473.316,A -85,B 0,C 180,E1 -16645.822,E2 -16645.822} C_VEL
LIN {X 0,Y 289.409,Z 474.49,A -85,B 0,C 180,E1 -16648.608,E2 -16648.608} C_VEL
LIN {X 0,Y 289.409,Z 474.486,A -85,B 0,C 180,E1 -16651.391,E2 -16651.391} C_VEL
LIN {X 0,Y 289.375,Z 473.298,A -85,B 0,C 180,E1 -16654.178,E2 -16654.178} C_VEL
LIN {X 0,Y 289.464,Z 470.953,A -85,B 0,C 180,E1 -16656.973,E2 -16656.973} C_VEL
LIN {X 0,Y 289.822,Z 467.404,A -85,B 0,C 180,E1 -16659.773,E2 -16659.773} C_VEL
LIN {X 0,Y 290.6,Z 462.565,A -85,B 0,C 180,E1 -16662.572,E2 -16662.572} C_VEL
LIN {X 0,Y 291.747,Z 455.926,A -85,B 0,C 180,E1 -16665.513,E2 -16665.513} C_VEL
LIN {X 0,Y 293.52,Z 448.449,A -85,B 0,C 180,E1 -16668.136,E2 -16668.136} C_VEL
LIN {X 0,Y 295.521,Z 440.103,A -85,B 0,C 180,E1 -16670.535,E2 -16670.535} C_VEL
LIN {X 0,Y 297.82,Z 430.963,A -85,B 0,C 180,E1 -16672.7,E2 -16672.7} C_VEL
LIN {X 0,Y 300.469,Z 419.783,A -85,B 0,C 180,E1 -16674.899,E2 -16674.899} C_VEL
LIN {X 0,Y 303.335,Z 407.546,A -85,B 0,C 180,E1 -16676.859,E2 -16676.859} C_VEL
LIN {X 0,Y 306.314,Z 393.923,A -85,B 0,C 180,E1 -16678.617,E2 -16678.617} C_VEL
LIN {X 0,Y 309.128,Z 379.445,A -85,B 0,C 180,E1 -16680.099,E2 -16680.099} C_VEL
LIN {X 0,Y 311.398,Z 364.987,A -85,B 0,C 180,E1 -16681.271,E2 -16681.271} C_VEL
LIN {X 0,Y 313.419,Z 350.04,A -85,B 0,C 180,E1 -16682.179,E2 -16682.179} C_VEL
LIN {X 0,Y 314.917,Z 335.521,A -85,B 0,C 180,E1 -16682.812,E2 -16682.812} C_VEL
LIN {X 0,Y 315.857,Z 319.421,A -85,B 0,C 180,E1 -16683.272,E2 -16683.272} C_VEL
LIN {X 0,Y 319.012,Z 235.381,A -85,B 0,C 180,E1 -16685.135,E2 -16685.135} C_VEL
LIN {X 0,Y 319.591,Z 217.398,A -85,B 0,C 180,E1 -16685.546,E2 -16685.546} C_VEL
LIN {X 0,Y 317.788,Z 207.329,A -85,B 0,C 180,E1 -16686.051,E2 -16686.051} C_VEL
LIN {X 0,Y 309.877,Z 189.73,A -85,B 0,C 180,E1 -16687.616,E2 -16687.616} C_VEL
LIN {X 0,Y 302.358,Z 174.873,A -85,B 0,C 180,E1 -16689.156,E2 -16689.156} C_VEL
LIN {X 0,Y 294.861,Z 161.255,A -85,B 0,C 180,E1 -16690.821,E2 -16690.821} C_VEL
LIN {X 0,Y 291.704,Z 151.363,A -85,B 0,C 180,E1 -16694.322,E2 -16694.322} C_VEL
LIN {X 0,Y 291.324,Z 149.818,A -85,B 0,C 180,E1 -16694.929,E2 -16694.929} C_VEL
LIN {X 0,Y 291.327,Z 149.818,A -85,B 0,C 180,E1 -16698.404,E2 -16698.404} C_VEL
LIN {X 0,Y 291.348,Z 149.813,A -85,B 0,C 180,E1 -16701.158,E2 -16701.158} C_VEL
LIN {X 0,Y 291.361,Z 149.809,A -85,B 0,C 180,E1 -16704.626,E2 -16704.626} C_VEL
LIN {X 0,Y 291.373,Z 149.812,A -85,B 0,C 180,E1 -16707.951,E2 -16707.951} C_VEL
LIN {X 0,Y 291.384,Z 149.811,A -85,B 0,C 180,E1 -16711.159,E2 -16711.159} C_VEL
LIN {X 0,Y 291.418,Z 149.808,A -85,B 0,C 180,E1 -16714.272,E2 -16714.272} C_VEL
LIN {X 0,Y 291.383,Z 149.811,A -85,B 0,C 180,E1 -16717.3,E2 -16717.3} C_VEL
LIN {X 0,Y 291.459,Z 149.796,A -85,B 0,C 180,E1 -16720.27,E2 -16720.27} C_VEL
LIN {X 0,Y 291.557,Z 149.787,A -85,B 0,C 180,E1 -16724.624,E2 -16724.624} C_VEL
LIN {X 0,Y 291.531,Z 149.793,A -85,B 0,C 180,E1 -16728.881,E2 -16728.881} C_VEL
LIN {X 0,Y 291.653,Z 149.77,A -85,B 0,C 180,E1 -16731.687,E2 -16731.687} C_VEL
LIN {X 0,Y 291.606,Z 149.785,A -85,B 0,C 180,E1 -16734.468,E2 -16734.468} C_VEL
LIN {X 0,Y 291.878,Z 149.751,A -85,B 0,C 180,E1 -16738.62,E2 -16738.62} C_VEL
LIN {X 0,Y 291.881,Z 149.749,A -85,B 0,C 180,E1 -16741.38,E2 -16741.38} C_VEL
LIN {X 0,Y 291.689,Z 149.776,A -85,B 0,C 180,E1 -16746.919,E2 -16746.919} C_VEL
LIN {X 0,Y 291.57,Z 149.783,A -85,B 0,C 180,E1 -16749.714,E2 -16749.714} C_VEL
LIN {X 0,Y 291.484,Z 149.795,A -85,B 0,C 180,E1 -16753.952,E2 -16753.952} C_VEL
LIN {X 0,Y 291.421,Z 149.806,A -85,B 0,C 180,E1 -16758.271,E2 -16758.271} C_VEL
LIN {X 0,Y 291.362,Z 149.808,A -85,B 0,C 180,E1 -16761.212,E2 -16761.212} C_VEL
LIN {X 0,Y 291.361,Z 149.81,A -85,B 0,C 180,E1 -16764.209,E2 -16764.209} C_VEL
LIN {X 0,Y 291.354,Z 149.789,A -85,B 0,C 180,E1 -16767.279,E2 -16767.279} C_VEL
LIN {X 0,Y 291.319,Z 149.821,A -85,B 0,C 180,E1 -16770.439,E2 -16770.439} C_VEL
LIN {X 0,Y 291.345,Z 149.814,A -85,B 0,C 180,E1 -16773.699,E2 -16773.699} C_VEL
LIN {X 0,Y 291.36,Z 149.811,A -85,B 0,C 180,E1 -16777.249,E2 -16777.249} C_VEL
LIN {X 0,Y 291.301,Z 149.82,A -85,B 0,C 180,E1 -16780.648,E2 -16780.648} C_VEL
LIN {X 0,Y 291.282,Z 149.822,A -85,B 0,C 180,E1 -16784.404,E2 -16784.404} C_VEL
LIN {X 0,Y 291.343,Z 149.964,A -85,B 0,C 180,E1 -16788.712,E2 -16788.712} C_VEL
LIN {X 0,Y 292.303,Z 152.668,A -85,B 0,C 180,E1 -16788.965,E2 -16788.965} C_VEL
LIN {X 0,Y 294.253,Z 155.09,A -85,B 0,C 180,E1 -16789.374,E2 -16789.374} C_VEL
LIN {X 0,Y 296.477,Z 158.487,A -85,B 0,C 180,E1 -16789.85,E2 -16789.85} C_VEL
LIN {X 0,Y 302.473,Z 168.246,A -85,B 0,C 180,E1 -16791.102,E2 -16791.102} C_VEL
LIN {X 0,Y 310.113,Z 182.503,A -85,B 0,C 180,E1 -16792.65,E2 -16792.65} C_VEL
LIN {X 0,Y 317.512,Z 197.951,A -85,B 0,C 180,E1 -16794.095,E2 -16794.095} C_VEL
LIN {X 0,Y 320.037,Z 203.735,A -85,B 0,C 180,E1 -16794.581,E2 -16794.581} C_VEL
LIN {X 0,Y 317.401,Z 276.675,A -85,B 0,C 180,E1 -16796.213,E2 -16796.213} C_VEL
LIN {X 0,Y 315.865,Z 313.885,A -85,B 0,C 180,E1 -16797.062,E2 -16797.062} C_VEL
LIN {X 0,Y 314.779,Z 328.195,A -85,B 0,C 180,E1 -16797.599,E2 -16797.599} C_VEL
LIN {X 0,Y 313.456,Z 340.993,A -85,B 0,C 180,E1 -16798.28,E2 -16798.28} C_VEL
LIN {X 0,Y 311.749,Z 354.23,A -85,B 0,C 180,E1 -16799.194,E2 -16799.194} C_VEL
LIN {X 0,Y 309.524,Z 368.08,A -85,B 0,C 180,E1 -16800.406,E2 -16800.406} C_VEL
LIN {X 0,Y 307.03,Z 381.138,A -85,B 0,C 180,E1 -16801.828,E2 -16801.828} C_VEL
LIN {X 0,Y 304.446,Z 393.158,A -85,B 0,C 180,E1 -16803.432,E2 -16803.432} C_VEL
LIN {X 0,Y 301.696,Z 404.701,A -85,B 0,C 180,E1 -16805.3,E2 -16805.3} C_VEL
LIN {X 0,Y 299.857,Z 412.819,A -85,B 0,C 180,E1 -16806.885,E2 -16806.885} C_VEL
LIN {X 0,Y 297.256,Z 423.052,A -85,B 0,C 180,E1 -16809.228,E2 -16809.228} C_VEL
LIN {X 0,Y 295.027,Z 431.546,A -85,B 0,C 180,E1 -16811.601,E2 -16811.601} C_VEL
LIN {X 0,Y 293.279,Z 438.609,A -85,B 0,C 180,E1 -16814.003,E2 -16814.003} C_VEL
LIN {X 0,Y 292.148,Z 443.669,A -85,B 0,C 180,E1 -16816.08,E2 -16816.08} C_VEL
LIN {X 0,Y 290.924,Z 449.112,A -85,B 0,C 180,E1 -16818.857,E2 -16818.857} C_VEL
LIN {X 0,Y 290.189,Z 453.216,A -85,B 0,C 180,E1 -16821.645,E2 -16821.645} C_VEL
LIN {X 0,Y 289.717,Z 456.099,A -85,B 0,C 180,E1 -16824.432,E2 -16824.432} C_VEL
LIN {X 0,Y 289.53,Z 457.83,A -85,B 0,C 180,E1 -16827.217,E2 -16827.217} C_VEL
LIN {X 0,Y 289.442,Z 458.435,A -85,B 0,C 180,E1 -16830,E2 -16830} C_VEL
LIN {X 0,Y 289.53,Z 457.871,A -85,B 0,C 180,E1 -16832.783,E2 -16832.783} C_VEL
LIN {X 0,Y 289.716,Z 456.195,A -85,B 0,C 180,E1 -16835.568,E2 -16835.568} C_VEL
LIN {X 0,Y 290.164,Z 453.364,A -85,B 0,C 180,E1 -16838.356,E2 -16838.356} C_VEL
LIN {X 0,Y 290.892,Z 449.311,A -85,B 0,C 180,E1 -16841.144,E2 -16841.144} C_VEL
LIN {X 0,Y 292.127,Z 443.93,A -85,B 0,C 180,E1 -16843.921,E2 -16843.921} C_VEL
LIN {X 0,Y 293.671,Z 437.074,A -85,B 0,C 180,E1 -16846.689,E2 -16846.689} C_VEL
LIN {X 0,Y 295.864,Z 428.507,A -85,B 0,C 180,E1 -16849.424,E2 -16849.424} C_VEL
LIN {X 0,Y 298.203,Z 419.395,A -85,B 0,C 180,E1 -16851.789,E2 -16851.789} C_VEL
LIN {X 0,Y 300.855,Z 409.171,A -85,B 0,C 180,E1 -16853.965,E2 -16853.965} C_VEL
LIN {X 0,Y 303.564,Z 397.031,A -85,B 0,C 180,E1 -16856.096,E2 -16856.096} C_VEL
LIN {X 0,Y 306.405,Z 384.528,A -85,B 0,C 180,E1 -16857.862,E2 -16857.862} C_VEL
LIN {X 0,Y 308.62,Z 373.706,A -85,B 0,C 180,E1 -16859.128,E2 -16859.128} C_VEL
LIN {X 0,Y 310.929,Z 360.021,A -85,B 0,C 180,E1 -16860.451,E2 -16860.451} C_VEL
LIN {X 0,Y 313.021,Z 345.066,A -85,B 0,C 180,E1 -16861.583,E2 -16861.583} C_VEL
LIN {X 0,Y 314.65,Z 330.269,A -85,B 0,C 180,E1 -16862.416,E2 -16862.416} C_VEL
LIN {X 0,Y 315.947,Z 314.51,A -85,B 0,C 180,E1 -16863.024,E2 -16863.024} C_VEL
LIN {X 0,Y 318.518,Z 249.17,A -85,B 0,C 180,E1 -16864.508,E2 -16864.508} C_VEL
LIN {X 0,Y 320.22,Z 203.977,A -85,B 0,C 180,E1 -16865.511,E2 -16865.511} C_VEL
LIN {X 0,Y 312.781,Z 187.668,A -85,B 0,C 180,E1 -16866.954,E2 -16866.954} C_VEL
LIN {X 0,Y 303.888,Z 170.63,A -85,B 0,C 180,E1 -16868.74,E2 -16868.74} C_VEL
LIN {X 0,Y 302.592,Z 168.468,A -85,B 0,C 180,E1 -16869.003,E2 -16869.003} C_VEL
LIN {X 0,Y 300.465,Z 165.942,A -85,B 0,C 180,E1 -16869.411,E2 -16869.411} C_VEL
LIN {X 0,Y 295.978,Z 163.301,A -85,B 0,C 180,E1 -16870.215,E2 -16870.215} C_VEL
LIN {X 0,Y 291.336,Z 160.932,A -85,B 0,C 180,E1 -16871.073,E2 -16871.073} C_VEL
LIN {X 0,Y 288.954,Z 158.781,A -85,B 0,C 180,E1 -16871.558,E2 -16871.558} C_VEL
LIN {X 0,Y 286.595,Z 155.151,A -85,B 0,C 180,E1 -16872.101,E2 -16872.101} C_VEL
LIN {X 0,Y 284.888,Z 152.859,A -85,B 0,C 180,E1 -16872.49,E2 -16872.49} C_VEL
LIN {X 0,Y 284.251,Z 150.702,A -85,B 0,C 180,E1 -16872.693,E2 -16872.693} C_VEL
LIN {X 0,Y 284.238,Z 150.696,A -85,B 0,C 180,E1 -16876.186,E2 -16876.186} C_VEL
LIN {X 0,Y 284.257,Z 150.703,A -85,B 0,C 180,E1 -16880.036,E2 -16880.036} C_VEL
LIN {X 0,Y 284.32,Z 150.673,A -85,B 0,C 180,E1 -16883.612,E2 -16883.612} C_VEL
LIN {X 0,Y 284.307,Z 150.677,A -85,B 0,C 180,E1 -16887.191,E2 -16887.191} C_VEL
LIN {X 0,Y 284.314,Z 150.677,A -85,B 0,C 180,E1 -16890.371,E2 -16890.371} C_VEL
LIN {X 0,Y 284.299,Z 150.689,A -85,B 0,C 180,E1 -16893.579,E2 -16893.579} C_VEL
LIN {X 0,Y 284.311,Z 150.691,A -85,B 0,C 180,E1 -16896.702,E2 -16896.702} C_VEL
LIN {X 0,Y 284.335,Z 150.693,A -85,B 0,C 180,E1 -16899.928,E2 -16899.928} C_VEL
LIN {X 0,Y 284.438,Z 150.678,A -85,B 0,C 180,E1 -16904.501,E2 -16904.501} C_VEL
LIN {X 0,Y 284.484,Z 150.673,A -85,B 0,C 180,E1 -16908.601,E2 -16908.601} C_VEL
LIN {X 0,Y 284.61,Z 150.647,A -85,B 0,C 180,E1 -16911.48,E2 -16911.48} C_VEL
LIN {X 0,Y 284.569,Z 150.656,A -85,B 0,C 180,E1 -16914.33,E2 -16914.33} C_VEL
LIN {X 0,Y 284.847,Z 150.626,A -85,B 0,C 180,E1 -16918.586,E2 -16918.586} C_VEL
LIN {X 0,Y 284.846,Z 150.623,A -85,B 0,C 180,E1 -16921.414,E2 -16921.414} C_VEL
LIN {X 0,Y 284.575,Z 150.655,A -85,B 0,C 180,E1 -16925.669,E2 -16925.669} C_VEL
LIN {X 0,Y 284.61,Z 150.649,A -85,B 0,C 180,E1 -16928.98,E2 -16928.98} C_VEL
LIN {X 0,Y 284.475,Z 150.671,A -85,B 0,C 180,E1 -16932.847,E2 -16932.847} C_VEL
LIN {X 0,Y 284.428,Z 150.684,A -85,B 0,C 180,E1 -16935.771,E2 -16935.771} C_VEL
LIN {X 0,Y 284.37,Z 150.691,A -85,B 0,C 180,E1 -16940.243,E2 -16940.243} C_VEL
LIN {X 0,Y 284.328,Z 150.695,A -85,B 0,C 180,E1 -16943.855,E2 -16943.855} C_VEL
LIN {X 0,Y 284.293,Z 150.698,A -85,B 0,C 180,E1 -16948.015,E2 -16948.015} C_VEL
LIN {X 0,Y 284.288,Z 150.698,A -85,B 0,C 180,E1 -16951.275,E2 -16951.275} C_VEL
LIN {X 0,Y 284.342,Z 150.692,A -85,B 0,C 180,E1 -16955.348,E2 -16955.348} C_VEL
LIN {X 0,Y 284.313,Z 150.694,A -85,B 0,C 180,E1 -16958.169,E2 -16958.169} C_VEL
LIN {X 0,Y 284.27,Z 150.696,A -85,B 0,C 180,E1 -16962.124,E2 -16962.124} C_VEL
LIN {X 0,Y 284.281,Z 150.856,A -85,B 0,C 180,E1 -16964.071,E2 -16964.071} C_VEL
LIN {X 0,Y 287.559,Z 161.227,A -85,B 0,C 180,E1 -16967.925,E2 -16967.925} C_VEL
LIN {X 0,Y 290.243,Z 165.83,A -85,B 0,C 180,E1 -16968.547,E2 -16968.547} C_VEL
LIN {X 0,Y 298.098,Z 179.988,A -85,B 0,C 180,E1 -16970.294,E2 -16970.294} C_VEL
LIN {X 0,Y 305.848,Z 195.551,A -85,B 0,C 180,E1 -16971.937,E2 -16971.937} C_VEL
LIN {X 0,Y 312.556,Z 210.83,A -85,B 0,C 180,E1 -16973.317,E2 -16973.317} C_VEL
LIN {X 0,Y 313.932,Z 219.891,A -85,B 0,C 180,E1 -16973.754,E2 -16973.754} C_VEL
LIN {X 0,Y 309.607,Z 327.976,A -85,B 0,C 180,E1 -16976.21,E2 -16976.21} C_VEL
LIN {X 0,Y 308.276,Z 343.383,A -85,B 0,C 180,E1 -16976.78,E2 -16976.78} C_VEL
LIN {X 0,Y 306.374,Z 358.284,A -85,B 0,C 180,E1 -16977.574,E2 -16977.574} C_VEL
LIN {X 0,Y 304.112,Z 372.984,A -85,B 0,C 180,E1 -16978.643,E2 -16978.643} C_VEL
LIN {X 0,Y 301.587,Z 386.722,A -85,B 0,C 180,E1 -16979.932,E2 -16979.932} C_VEL
LIN {X 0,Y 298.635,Z 400.446,A -85,B 0,C 180,E1 -16981.539,E2 -16981.539} C_VEL
LIN {X 0,Y 295.682,Z 412.875,A -85,B 0,C 180,E1 -16983.344,E2 -16983.344} C_VEL
LIN {X 0,Y 292.692,Z 425.07,A -85,B 0,C 180,E1 -16985.531,E2 -16985.531} C_VEL
LIN {X 0,Y 290.012,Z 435.923,A -85,B 0,C 180,E1 -16987.937,E2 -16987.937} C_VEL
LIN {X 0,Y 287.58,Z 444.962,A -85,B 0,C 180,E1 -16990.365,E2 -16990.365} C_VEL
LIN {X 0,Y 285.486,Z 453.527,A -85,B 0,C 180,E1 -16993.223,E2 -16993.223} C_VEL
LIN {X 0,Y 284.173,Z 459.478,A -85,B 0,C 180,E1 -16995.681,E2 -16995.681} C_VEL
LIN {X 0,Y 283.087,Z 464.992,A -85,B 0,C 180,E1 -16998.544,E2 -16998.544} C_VEL
LIN {X 0,Y 282.551,Z 469.168,A -85,B 0,C 180,E1 -17001.417,E2 -17001.417} C_VEL
LIN {X 0,Y 282.348,Z 472.392,A -85,B 0,C 180,E1 -17004.653,E2 -17004.653} C_VEL
LIN {X 0,Y 282.323,Z 473.848,A -85,B 0,C 180,E1 -17007.146,E2 -17007.146} C_VEL
LIN {X 0,Y 282.354,Z 474.446,A -85,B 0,C 180,E1 -17010,E2 -17010} C_VEL
LIN {X 0,Y 282.323,Z 473.837,A -85,B 0,C 180,E1 -17012.854,E2 -17012.854} C_VEL
LIN {X 0,Y 282.335,Z 472.074,A -85,B 0,C 180,E1 -17015.714,E2 -17015.714} C_VEL
LIN {X 0,Y 282.551,Z 469.134,A -85,B 0,C 180,E1 -17018.583,E2 -17018.583} C_VEL
LIN {X 0,Y 283.084,Z 464.95,A -85,B 0,C 180,E1 -17021.456,E2 -17021.456} C_VEL
LIN {X 0,Y 284.152,Z 459.418,A -85,B 0,C 180,E1 -17024.32,E2 -17024.32} C_VEL
LIN {X 0,Y 285.248,Z 454.274,A -85,B 0,C 180,E1 -17026.46,E2 -17026.46} C_VEL
LIN {X 0,Y 286.981,Z 447.122,A -85,B 0,C 180,E1 -17028.934,E2 -17028.934} C_VEL
LIN {X 0,Y 289.236,Z 438.541,A -85,B 0,C 180,E1 -17031.375,E2 -17031.375} C_VEL
LIN {X 0,Y 291.709,Z 428.555,A -85,B 0,C 180,E1 -17033.722,E2 -17033.722} C_VEL
LIN {X 0,Y 294.45,Z 417.659,A -85,B 0,C 180,E1 -17035.823,E2 -17035.823} C_VEL
LIN {X 0,Y 297.234,Z 406.187,A -85,B 0,C 180,E1 -17037.647,E2 -17037.647} C_VEL
LIN {X 0,Y 300.091,Z 393.72,A -85,B 0,C 180,E1 -17039.267,E2 -17039.267} C_VEL
LIN {X 0,Y 302.831,Z 380.062,A -85,B 0,C 180,E1 -17040.702,E2 -17040.702} C_VEL
LIN {X 0,Y 305.173,Z 365.91,A -85,B 0,C 180,E1 -17041.887,E2 -17041.887} C_VEL
LIN {X 0,Y 307.344,Z 350.595,A -85,B 0,C 180,E1 -17042.845,E2 -17042.845} C_VEL
LIN {X 0,Y 308.98,Z 335.309,A -85,B 0,C 180,E1 -17043.525,E2 -17043.525} C_VEL
LIN {X 0,Y 309.939,Z 319.201,A -85,B 0,C 180,E1 -17043.993,E2 -17043.993} C_VEL
LIN {X 0,Y 313.237,Z 234.931,A -85,B 0,C 180,E1 -17045.888,E2 -17045.888} C_VEL
LIN {X 0,Y 313.792,Z 218.659,A -85,B 0,C 180,E1 -17046.265,E2 -17046.265} C_VEL
LIN {X 0,Y 312.305,Z 210.244,A -85,B 0,C 180,E1 -17046.699,E2 -17046.699} C_VEL
LIN {X 0,Y 303.73,Z 191.09,A -85,B 0,C 180,E1 -17048.467,E2 -17048.467} C_VEL
LIN {X 0,Y 295.469,Z 175.153,A -85,B 0,C 180,E1 -17050.235,E2 -17050.235} C_VEL
LIN {X 0,Y 289.788,Z 165.241,A -85,B 0,C 180,E1 -17051.504,E2 -17051.504} C_VEL
LIN {X 0,Y 287.468,Z 160.98,A -85,B 0,C 180,E1 -17052.106,E2 -17052.106} C_VEL
LIN {X 0,Y 284.257,Z 150.701,A -85,B 0,C 180,E1 -17055.991,E2 -17055.991} C_VEL
LIN {X 0,Y 284.307,Z 150.694,A -85,B 0,C 180,E1 -17060.024,E2 -17060.024} C_VEL
LIN {X 0,Y 284.331,Z 150.685,A -85,B 0,C 180,E1 -17063.614,E2 -17063.614} C_VEL
LIN {X 0,Y 284.309,Z 150.687,A -85,B 0,C 180,E1 -17067.19,E2 -17067.19} C_VEL
LIN {X 0,Y 284.36,Z 150.681,A -85,B 0,C 180,E1 -17070.376,E2 -17070.376} C_VEL
LIN {X 0,Y 284.379,Z 150.681,A -85,B 0,C 180,E1 -17073.587,E2 -17073.587} C_VEL
LIN {X 0,Y 284.367,Z 150.681,A -85,B 0,C 180,E1 -17076.707,E2 -17076.707} C_VEL
LIN {X 0,Y 284.406,Z 150.683,A -85,B 0,C 180,E1 -17081.262,E2 -17081.262} C_VEL
LIN {X 0,Y 284.494,Z 150.666,A -85,B 0,C 180,E1 -17084.459,E2 -17084.459} C_VEL
LIN {X 0,Y 284.485,Z 150.668,A -85,B 0,C 180,E1 -17088.601,E2 -17088.601} C_VEL
LIN {X 0,Y 284.61,Z 150.647,A -85,B 0,C 180,E1 -17091.48,E2 -17091.48} C_VEL
LIN {X 0,Y 284.575,Z 150.662,A -85,B 0,C 180,E1 -17094.331,E2 -17094.331} C_VEL
LIN {X 0,Y 284.845,Z 150.628,A -85,B 0,C 180,E1 -17098.586,E2 -17098.586} C_VEL
LIN {X 0,Y 284.847,Z 150.625,A -85,B 0,C 180,E1 -17101.414,E2 -17101.414} C_VEL
LIN {X 0,Y 284.645,Z 150.653,A -85,B 0,C 180,E1 -17107.092,E2 -17107.092} C_VEL
LIN {X 0,Y 284.515,Z 150.663,A -85,B 0,C 180,E1 -17109.957,E2 -17109.957} C_VEL
LIN {X 0,Y 284.436,Z 150.676,A -85,B 0,C 180,E1 -17114.305,E2 -17114.305} C_VEL
LIN {X 0,Y 284.369,Z 150.687,A -85,B 0,C 180,E1 -17118.741,E2 -17118.741} C_VEL
LIN {X 0,Y 284.317,Z 150.688,A -85,B 0,C 180,E1 -17121.764,E2 -17121.764} C_VEL
LIN {X 0,Y 284.306,Z 150.677,A -85,B 0,C 180,E1 -17124.85,E2 -17124.85} C_VEL
LIN {X 0,Y 284.284,Z 150.679,A -85,B 0,C 180,E1 -17128.016,E2 -17128.016} C_VEL
LIN {X 0,Y 284.286,Z 150.693,A -85,B 0,C 180,E1 -17131.276,E2 -17131.276} C_VEL
LIN {X 0,Y 284.338,Z 150.689,A -85,B 0,C 180,E1 -17135.347,E2 -17135.347} C_VEL
LIN {X 0,Y 284.299,Z 150.694,A -85,B 0,C 180,E1 -17138.171,E2 -17138.171} C_VEL
LIN {X 0,Y 284.238,Z 150.697,A -85,B 0,C 180,E1 -17142.117,E2 -17142.117} C_VEL
LIN {X 0,Y 284.238,Z 150.702,A -85,B 0,C 180,E1 -17146.186,E2 -17146.186} C_VEL
LIN {X 0,Y 284.283,Z 150.891,A -85,B 0,C 180,E1 -17147.471,E2 -17147.471} C_VEL
LIN {X 0,Y 285.204,Z 153.494,A -85,B 0,C 180,E1 -17147.729,E2 -17147.729} C_VEL
LIN {X 0,Y 287.286,Z 156.083,A -85,B 0,C 180,E1 -17148.194,E2 -17148.194} C_VEL
LIN {X 0,Y 289.628,Z 159.555,A -85,B 0,C 180,E1 -17148.722,E2 -17148.722} C_VEL
LIN {X 0,Y 296.403,Z 170.186,A -85,B 0,C 180,E1 -17150.201,E2 -17150.201} C_VEL
LIN {X 0,Y 303.818,Z 183.703,A -85,B 0,C 180,E1 -17151.766,E2 -17151.766} C_VEL
LIN {X 0,Y 311.654,Z 199.988,A -85,B 0,C 180,E1 -17153.362,E2 -17153.362} C_VEL
LIN {X 0,Y 314.271,Z 206.019,A -85,B 0,C 180,E1 -17153.887,E2 -17153.887} C_VEL
LIN {X 0,Y 309.95,Z 314.1,A -85,B 0,C 180,E1 -17156.35,E2 -17156.35} C_VEL
LIN {X 0,Y 308.779,Z 328.907,A -85,B 0,C 180,E1 -17156.916,E2 -17156.916} C_VEL
LIN {X 0,Y 307.329,Z 342.367,A -85,B 0,C 180,E1 -17157.658,E2 -17157.658} C_VEL
LIN {X 0,Y 305.583,Z 355.029,A -85,B 0,C 180,E1 -17158.56,E2 -17158.56} C_VEL
LIN {X 0,Y 303.381,Z 368.284,A -85,B 0,C 180,E1 -17159.745,E2 -17159.745} C_VEL
LIN {X 0,Y 300.777,Z 381.342,A -85,B 0,C 180,E1 -17161.189,E2 -17161.189} C_VEL
LIN {X 0,Y 298.119,Z 393.361,A -85,B 0,C 180,E1 -17162.822,E2 -17162.822} C_VEL
LIN {X 0,Y 295.383,Z 404.462,A -85,B 0,C 180,E1 -17164.642,E2 -17164.642} C_VEL
LIN {X 0,Y 292.877,Z 414.64,A -85,B 0,C 180,E1 -17166.675,E2 -17166.675} C_VEL
LIN {X 0,Y 290.245,Z 424.598,A -85,B 0,C 180,E1 -17169.074,E2 -17169.074} C_VEL
LIN {X 0,Y 287.964,Z 432.856,A -85,B 0,C 180,E1 -17171.502,E2 -17171.502} C_VEL
LIN {X 0,Y 286.397,Z 438.811,A -85,B 0,C 180,E1 -17173.608,E2 -17173.608} C_VEL
LIN {X 0,Y 285.248,Z 443.87,A -85,B 0,C 180,E1 -17175.736,E2 -17175.736} C_VEL
LIN {X 0,Y 283.923,Z 449.313,A -85,B 0,C 180,E1 -17178.578,E2 -17178.578} C_VEL
LIN {X 0,Y 283.146,Z 453.416,A -85,B 0,C 180,E1 -17181.435,E2 -17181.435} C_VEL
LIN {X 0,Y 282.651,Z 456.298,A -85,B 0,C 180,E1 -17184.292,E2 -17184.292} C_VEL
LIN {X 0,Y 282.461,Z 458.028,A -85,B 0,C 180,E1 -17187.148,E2 -17187.148} C_VEL
LIN {X 0,Y 282.361,Z 458.633,A -85,B 0,C 180,E1 -17190,E2 -17190} C_VEL
LIN {X 0,Y 282.461,Z 458.069,A -85,B 0,C 180,E1 -17192.852,E2 -17192.852} C_VEL
LIN {X 0,Y 282.711,Z 456.105,A -85,B 0,C 180,E1 -17196.079,E2 -17196.079} C_VEL
LIN {X 0,Y 283.126,Z 453.563,A -85,B 0,C 180,E1 -17198.565,E2 -17198.565} C_VEL
LIN {X 0,Y 283.892,Z 449.51,A -85,B 0,C 180,E1 -17201.423,E2 -17201.423} C_VEL
LIN {X 0,Y 285.221,Z 444.128,A -85,B 0,C 180,E1 -17204.265,E2 -17204.265} C_VEL
LIN {X 0,Y 286.926,Z 436.979,A -85,B 0,C 180,E1 -17207.201,E2 -17207.201} C_VEL
LIN {X 0,Y 289.131,Z 428.705,A -85,B 0,C 180,E1 -17209.895,E2 -17209.895} C_VEL
LIN {X 0,Y 291.595,Z 419.592,A -85,B 0,C 180,E1 -17212.309,E2 -17212.309} C_VEL
LIN {X 0,Y 294.281,Z 409.632,A -85,B 0,C 180,E1 -17214.479,E2 -17214.479} C_VEL
LIN {X 0,Y 297.175,Z 397.227,A -85,B 0,C 180,E1 -17216.701,E2 -17216.701} C_VEL
LIN {X 0,Y 299.885,Z 386,A -85,B 0,C 180,E1 -17218.332,E2 -17218.332} C_VEL
LIN {X 0,Y 302.127,Z 375.321,A -85,B 0,C 180,E1 -17219.625,E2 -17219.625} C_VEL
LIN {X 0,Y 304.569,Z 361.938,A -85,B 0,C 180,E1 -17220.968,E2 -17220.968} C_VEL
LIN {X 0,Y 306.572,Z 348.492,A -85,B 0,C 180,E1 -17222.048,E2 -17222.048} C_VEL
LIN {X 0,Y 308.345,Z 333.804,A -85,B 0,C 180,E1 -17222.949,E2 -17222.949} C_VEL
LIN {X 0,Y 309.667,Z 319.248,A -85,B 0,C 180,E1 -17223.587,E2 -17223.587} C_VEL
LIN {X 0,Y 310.622,Z 302.272,A -85,B 0,C 180,E1 -17224.055,E2 -17224.055} C_VEL
LIN {X 0,Y 314.383,Z 206.117,A -85,B 0,C 180,E1 -17226.219,E2 -17226.219} C_VEL
LIN {X 0,Y 307.019,Z 190.035,A -85,B 0,C 180,E1 -17227.704,E2 -17227.704} C_VEL
LIN {X 0,Y 298.956,Z 174.559,A -85,B 0,C 180,E1 -17229.387,E2 -17229.387} C_VEL
LIN {X 0,Y 293.427,Z 165.412,A -85,B 0,C 180,E1 -17230.574,E2 -17230.574} C_VEL
LIN {X 0,Y 288.954,Z 158.781,A -85,B 0,C 180,E1 -17231.558,E2 -17231.558} C_VEL
LIN {X 0,Y 287.484,Z 157.746,A -85,B 0,C 180,E1 -17231.854,E2 -17231.854} C_VEL
LIN {X 0,Y 281,Z 157.013,A -85,B 0,C 180,E1 -17233.082,E2 -17233.082} C_VEL
LIN {X 0,Y 279.984,Z 156.375,A -85,B 0,C 180,E1 -17233.301,E2 -17233.301} C_VEL
LIN {X 0,Y 278.107,Z 154.273,A -85,B 0,C 180,E1 -17233.742,E2 -17233.742} C_VEL
LIN {X 0,Y 277.204,Z 151.579,A -85,B 0,C 180,E1 -17234.05,E2 -17234.05} C_VEL
LIN {X 0,Y 277.193,Z 151.562,A -85,B 0,C 180,E1 -17237.331,E2 -17237.331} C_VEL
LIN {X 0,Y 277.225,Z 151.556,A -85,B 0,C 180,E1 -17241.803,E2 -17241.803} C_VEL
LIN {X 0,Y 277.278,Z 151.56,A -85,B 0,C 180,E1 -17244.34,E2 -17244.34} C_VEL
LIN {X 0,Y 277.238,Z 151.548,A -85,B 0,C 180,E1 -17247.835,E2 -17247.835} C_VEL
LIN {X 0,Y 277.221,Z 151.572,A -85,B 0,C 180,E1 -17251.205,E2 -17251.205} C_VEL
LIN {X 0,Y 277.236,Z 151.569,A -85,B 0,C 180,E1 -17254.472,E2 -17254.472} C_VEL
LIN {X 0,Y 277.25,Z 151.565,A -85,B 0,C 180,E1 -17257.652,E2 -17257.652} C_VEL
LIN {X 0,Y 277.281,Z 151.567,A -85,B 0,C 180,E1 -17260.761,E2 -17260.761} C_VEL
LIN {X 0,Y 277.405,Z 151.549,A -85,B 0,C 180,E1 -17265.324,E2 -17265.324} C_VEL
LIN {X 0,Y 277.46,Z 151.541,A -85,B 0,C 180,E1 -17269.787,E2 -17269.787} C_VEL
LIN {X 0,Y 277.602,Z 151.53,A -85,B 0,C 180,E1 -17272.728,E2 -17272.728} C_VEL
LIN {X 0,Y 277.813,Z 151.502,A -85,B 0,C 180,E1 -17278.55,E2 -17278.55} C_VEL
LIN {X 0,Y 277.813,Z 151.5,A -85,B 0,C 180,E1 -17281.449,E2 -17281.449} C_VEL
LIN {X 0,Y 277.545,Z 151.531,A -85,B 0,C 180,E1 -17285.813,E2 -17285.813} C_VEL
LIN {X 0,Y 277.563,Z 151.526,A -85,B 0,C 180,E1 -17289.068,E2 -17289.068} C_VEL
LIN {X 0,Y 277.411,Z 151.547,A -85,B 0,C 180,E1 -17293.18,E2 -17293.18} C_VEL
LIN {X 0,Y 277.365,Z 151.563,A -85,B 0,C 180,E1 -17296.184,E2 -17296.184} C_VEL
LIN {X 0,Y 277.339,Z 151.567,A -85,B 0,C 180,E1 -17300.345,E2 -17300.345} C_VEL
LIN {X 0,Y 277.284,Z 151.572,A -85,B 0,C 180,E1 -17304.153,E2 -17304.153} C_VEL
LIN {X 0,Y 277.282,Z 151.568,A -85,B 0,C 180,E1 -17307.487,E2 -17307.487} C_VEL
LIN {X 0,Y 277.249,Z 151.576,A -85,B 0,C 180,E1 -17310.472,E2 -17310.472} C_VEL
LIN {X 0,Y 277.248,Z 151.565,A -85,B 0,C 180,E1 -17313.895,E2 -17313.895} C_VEL
LIN {X 0,Y 277.269,Z 151.565,A -85,B 0,C 180,E1 -17317.469,E2 -17317.469} C_VEL
LIN {X 0,Y 277.21,Z 151.581,A -85,B 0,C 180,E1 -17321.236,E2 -17321.236} C_VEL
LIN {X 0,Y 277.189,Z 151.582,A -85,B 0,C 180,E1 -17322.877,E2 -17322.877} C_VEL
LIN {X 0,Y 280.303,Z 161.206,A -85,B 0,C 180,E1 -17326.579,E2 -17326.579} C_VEL
LIN {X 0,Y 283.051,Z 165.736,A -85,B 0,C 180,E1 -17327.253,E2 -17327.253} C_VEL
LIN {X 0,Y 291.207,Z 180.08,A -85,B 0,C 180,E1 -17329.169,E2 -17329.169} C_VEL
LIN {X 0,Y 299.211,Z 195.803,A -85,B 0,C 180,E1 -17330.949,E2 -17330.949} C_VEL
LIN {X 0,Y 306.904,Z 213.194,A -85,B 0,C 180,E1 -17332.6,E2 -17332.6} C_VEL
LIN {X 0,Y 308.192,Z 220.725,A -85,B 0,C 180,E1 -17332.997,E2 -17332.997} C_VEL
LIN {X 0,Y 303.728,Z 327.794,A -85,B 0,C 180,E1 -17335.465,E2 -17335.465} C_VEL
LIN {X 0,Y 302.271,Z 344.024,A -85,B 0,C 180,E1 -17336.081,E2 -17336.081} C_VEL
LIN {X 0,Y 300.226,Z 359.3,A -85,B 0,C 180,E1 -17336.926,E2 -17336.926} C_VEL
LIN {X 0,Y 297.882,Z 373.791,A -85,B 0,C 180,E1 -17338.017,E2 -17338.017} C_VEL
LIN {X 0,Y 295.125,Z 388.033,A -85,B 0,C 180,E1 -17339.401,E2 -17339.401} C_VEL
LIN {X 0,Y 292.088,Z 401.46,A -85,B 0,C 180,E1 -17341.038,E2 -17341.038} C_VEL
LIN {X 0,Y 289.037,Z 413.692,A -85,B 0,C 180,E1 -17342.876,E2 -17342.876} C_VEL
LIN {X 0,Y 286.179,Z 424.871,A -85,B 0,C 180,E1 -17344.936,E2 -17344.936} C_VEL
LIN {X 0,Y 283.391,Z 435.724,A -85,B 0,C 180,E1 -17347.394,E2 -17347.394} C_VEL
LIN {X 0,Y 280.831,Z 444.763,A -85,B 0,C 180,E1 -17349.873,E2 -17349.873} C_VEL
LIN {X 0,Y 278.857,Z 452.269,A -85,B 0,C 180,E1 -17352.396,E2 -17352.396} C_VEL
LIN {X 0,Y 277.234,Z 459.279,A -85,B 0,C 180,E1 -17355.315,E2 -17355.315} C_VEL
LIN {X 0,Y 276.073,Z 464.793,A -85,B 0,C 180,E1 -17358.249,E2 -17358.249} C_VEL
LIN {X 0,Y 275.473,Z 468.969,A -85,B 0,C 180,E1 -17361.195,E2 -17361.195} C_VEL
LIN {X 0,Y 275.234,Z 471.9,A -85,B 0,C 180,E1 -17364.138,E2 -17364.138} C_VEL
LIN {X 0,Y 275.231,Z 473.649,A -85,B 0,C 180,E1 -17367.073,E2 -17367.073} C_VEL
LIN {X 0,Y 275.276,Z 474.248,A -85,B 0,C 180,E1 -17370,E2 -17370} C_VEL
LIN {X 0,Y 275.231,Z 473.638,A -85,B 0,C 180,E1 -17372.927,E2 -17372.927} C_VEL
LIN {X 0,Y 275.234,Z 471.873,A -85,B 0,C 180,E1 -17375.862,E2 -17375.862} C_VEL
LIN {X 0,Y 275.473,Z 468.933,A -85,B 0,C 180,E1 -17378.805,E2 -17378.805} C_VEL
LIN {X 0,Y 276.07,Z 464.749,A -85,B 0,C 180,E1 -17381.751,E2 -17381.751} C_VEL
LIN {X 0,Y 277.208,Z 459.216,A -85,B 0,C 180,E1 -17384.686,E2 -17384.686} C_VEL
LIN {X 0,Y 278.384,Z 454.072,A -85,B 0,C 180,E1 -17386.877,E2 -17386.877} C_VEL
LIN {X 0,Y 280.196,Z 446.919,A -85,B 0,C 180,E1 -17389.411,E2 -17389.411} C_VEL
LIN {X 0,Y 282.557,Z 438.337,A -85,B 0,C 180,E1 -17391.907,E2 -17391.907} C_VEL
LIN {X 0,Y 284.964,Z 429.09,A -85,B 0,C 180,E1 -17394.144,E2 -17394.144} C_VEL
LIN {X 0,Y 287.537,Z 419.377,A -85,B 0,C 180,E1 -17396.101,E2 -17396.101} C_VEL
LIN {X 0,Y 290.644,Z 407.139,A -85,B 0,C 180,E1 -17398.133,E2 -17398.133} C_VEL
LIN {X 0,Y 293.896,Z 393.516,A -85,B 0,C 180,E1 -17399.946,E2 -17399.946} C_VEL
LIN {X 0,Y 296.693,Z 379.856,A -85,B 0,C 180,E1 -17401.408,E2 -17401.408} C_VEL
LIN {X 0,Y 299.148,Z 365.704,A -85,B 0,C 180,E1 -17402.607,E2 -17402.607} C_VEL
LIN {X 0,Y 301.407,Z 350.387,A -85,B 0,C 180,E1 -17403.577,E2 -17403.577} C_VEL
LIN {X 0,Y 303.076,Z 335.096,A -85,B 0,C 180,E1 -17404.267,E2 -17404.267} C_VEL
LIN {X 0,Y 304.085,Z 318.981,A -85,B 0,C 180,E1 -17404.74,E2 -17404.74} C_VEL
LIN {X 0,Y 307.421,Z 237.636,A -85,B 0,C 180,E1 -17406.593,E2 -17406.593} C_VEL
LIN {X 0,Y 308.053,Z 219.794,A -85,B 0,C 180,E1 -17407.013,E2 -17407.013} C_VEL
LIN {X 0,Y 306.757,Z 212.853,A -85,B 0,C 180,E1 -17407.394,E2 -17407.394} C_VEL
LIN {X 0,Y 298.531,Z 194.458,A -85,B 0,C 180,E1 -17409.156,E2 -17409.156} C_VEL
LIN {X 0,Y 290.865,Z 179.551,A -85,B 0,C 180,E1 -17410.861,E2 -17410.861} C_VEL
LIN {X 0,Y 285.214,Z 169.575,A -85,B 0,C 180,E1 -17412.172,E2 -17412.172} C_VEL
LIN {X 0,Y 281.981,Z 164.275,A -85,B 0,C 180,E1 -17412.945,E2 -17412.945} C_VEL
LIN {X 0,Y 280.125,Z 160.804,A -85,B 0,C 180,E1 -17413.448,E2 -17413.448} C_VEL
LIN {X 0,Y 277.191,Z 151.577,A -85,B 0,C 180,E1 -17417.123,E2 -17417.123} C_VEL
LIN {X 0,Y 277.233,Z 151.574,A -85,B 0,C 180,E1 -17420.672,E2 -17420.672} C_VEL
LIN {X 0,Y 277.284,Z 151.561,A -85,B 0,C 180,E1 -17424.342,E2 -17424.342} C_VEL
LIN {X 0,Y 277.246,Z 151.57,A -85,B 0,C 180,E1 -17427.837,E2 -17427.837} C_VEL
LIN {X 0,Y 277.291,Z 151.567,A -85,B 0,C 180,E1 -17431.213,E2 -17431.213} C_VEL
LIN {X 0,Y 277.315,Z 151.565,A -85,B 0,C 180,E1 -17434.48,E2 -17434.48} C_VEL
LIN {X 0,Y 277.287,Z 151.57,A -85,B 0,C 180,E1 -17437.655,E2 -17437.655} C_VEL
LIN {X 0,Y 277.347,Z 151.557,A -85,B 0,C 180,E1 -17440.767,E2 -17440.767} C_VEL
LIN {X 0,Y 277.436,Z 151.552,A -85,B 0,C 180,E1 -17445.326,E2 -17445.326} C_VEL
LIN {X 0,Y 277.459,Z 151.548,A -85,B 0,C 180,E1 -17449.787,E2 -17449.787} C_VEL
LIN {X 0,Y 277.603,Z 151.525,A -85,B 0,C 180,E1 -17452.728,E2 -17452.728} C_VEL
LIN {X 0,Y 277.693,Z 151.516,A -85,B 0,C 180,E1 -17457.099,E2 -17457.099} C_VEL
LIN {X 0,Y 277.797,Z 151.497,A -85,B 0,C 180,E1 -17460,E2 -17460} C_VEL
LIN {X 0,Y 277.651,Z 151.523,A -85,B 0,C 180,E1 -17462.902,E2 -17462.902} C_VEL
LIN {X 0,Y 277.603,Z 151.53,A -85,B 0,C 180,E1 -17467.272,E2 -17467.272} C_VEL
LIN {X 0,Y 277.458,Z 151.545,A -85,B 0,C 180,E1 -17470.213,E2 -17470.213} C_VEL
LIN {X 0,Y 277.388,Z 151.558,A -85,B 0,C 180,E1 -17474.677,E2 -17474.677} C_VEL
LIN {X 0,Y 277.321,Z 151.566,A -85,B 0,C 180,E1 -17479.236,E2 -17479.236} C_VEL
LIN {X 0,Y 277.283,Z 151.565,A -85,B 0,C 180,E1 -17483.925,E2 -17483.925} C_VEL
LIN {X 0,Y 277.27,Z 151.544,A -85,B 0,C 180,E1 -17487.482,E2 -17487.482} C_VEL
LIN {X 0,Y 277.249,Z 151.573,A -85,B 0,C 180,E1 -17490.473,E2 -17490.473} C_VEL
LIN {X 0,Y 277.247,Z 151.569,A -85,B 0,C 180,E1 -17493.896,E2 -17493.896} C_VEL
LIN {X 0,Y 277.255,Z 151.567,A -85,B 0,C 180,E1 -17497.471,E2 -17497.471} C_VEL
LIN {X 0,Y 277.185,Z 151.581,A -85,B 0,C 180,E1 -17501.241,E2 -17501.241} C_VEL
LIN {X 0,Y 277.175,Z 151.581,A -85,B 0,C 180,E1 -17505.232,E2 -17505.232} C_VEL
LIN {X 0,Y 277.208,Z 151.664,A -85,B 0,C 180,E1 -17506.132,E2 -17506.132} C_VEL
LIN {X 0,Y 278.19,Z 154.392,A -85,B 0,C 180,E1 -17506.423,E2 -17506.423} C_VEL
LIN {X 0,Y 280.324,Z 156.999,A -85,B 0,C 180,E1 -17506.929,E2 -17506.929} C_VEL
LIN {X 0,Y 282.401,Z 160.182,A -85,B 0,C 180,E1 -17507.433,E2 -17507.433} C_VEL
LIN {X 0,Y 290.078,Z 171.688,A -85,B 0,C 180,E1 -17509.192,E2 -17509.192} C_VEL
LIN {X 0,Y 296.751,Z 183.428,A -85,B 0,C 180,E1 -17510.666,E2 -17510.666} C_VEL
LIN {X 0,Y 305.244,Z 200.728,A -85,B 0,C 180,E1 -17512.477,E2 -17512.477} C_VEL
LIN {X 0,Y 308.487,Z 208.06,A -85,B 0,C 180,E1 -17513.151,E2 -17513.151} C_VEL
LIN {X 0,Y 304.084,Z 314.314,A -85,B 0,C 180,E1 -17515.612,E2 -17515.612} C_VEL
LIN {X 0,Y 302.865,Z 329.117,A -85,B 0,C 180,E1 -17516.184,E2 -17516.184} C_VEL
LIN {X 0,Y 301.347,Z 342.575,A -85,B 0,C 180,E1 -17516.935,E2 -17516.935} C_VEL
LIN {X 0,Y 299.482,Z 355.72,A -85,B 0,C 180,E1 -17517.892,E2 -17517.892} C_VEL
LIN {X 0,Y 297.272,Z 368.488,A -85,B 0,C 180,E1 -17519.056,E2 -17519.056} C_VEL
LIN {X 0,Y 294.538,Z 381.546,A -85,B 0,C 180,E1 -17520.519,E2 -17520.519} C_VEL
LIN {X 0,Y 291.793,Z 393.564,A -85,B 0,C 180,E1 -17522.182,E2 -17522.182} C_VEL
LIN {X 0,Y 288.966,Z 404.664,A -85,B 0,C 180,E1 -17524.037,E2 -17524.037} C_VEL
LIN {X 0,Y 286.365,Z 414.842,A -85,B 0,C 180,E1 -17526.112,E2 -17526.112} C_VEL
LIN {X 0,Y 283.598,Z 424.8,A -85,B 0,C 180,E1 -17528.56,E2 -17528.56} C_VEL
LIN {X 0,Y 281.202,Z 433.057,A -85,B 0,C 180,E1 -17531.04,E2 -17531.04} C_VEL
LIN {X 0,Y 279.531,Z 439.072,A -85,B 0,C 180,E1 -17533.219,E2 -17533.219} C_VEL
LIN {X 0,Y 277.897,Z 445.559,A -85,B 0,C 180,E1 -17536.098,E2 -17536.098} C_VEL
LIN {X 0,Y 276.686,Z 450.673,A -85,B 0,C 180,E1 -17539.018,E2 -17539.018} C_VEL
LIN {X 0,Y 276.122,Z 453.616,A -85,B 0,C 180,E1 -17541.216,E2 -17541.216} C_VEL
LIN {X 0,Y 275.576,Z 456.498,A -85,B 0,C 180,E1 -17544.145,E2 -17544.145} C_VEL
LIN {X 0,Y 275.394,Z 458.226,A -85,B 0,C 180,E1 -17547.074,E2 -17547.074} C_VEL
LIN {X 0,Y 275.283,Z 458.831,A -85,B 0,C 180,E1 -17550,E2 -17550} C_VEL
LIN {X 0,Y 275.394,Z 458.267,A -85,B 0,C 180,E1 -17552.926,E2 -17552.926} C_VEL
LIN {X 0,Y 275.612,Z 456.467,A -85,B 0,C 180,E1 -17556.019,E2 -17556.019} C_VEL
LIN {X 0,Y 276.083,Z 453.762,A -85,B 0,C 180,E1 -17558.786,E2 -17558.786} C_VEL
LIN {X 0,Y 276.911,Z 449.708,A -85,B 0,C 180,E1 -17561.715,E2 -17561.715} C_VEL
LIN {X 0,Y 278.307,Z 444.327,A -85,B 0,C 180,E1 -17564.627,E2 -17564.627} C_VEL
LIN {X 0,Y 280.026,Z 437.471,A -85,B 0,C 180,E1 -17567.528,E2 -17567.528} C_VEL
LIN {X 0,Y 282.433,Z 428.903,A -85,B 0,C 180,E1 -17570.388,E2 -17570.388} C_VEL
LIN {X 0,Y 285.018,Z 419.789,A -85,B 0,C 180,E1 -17572.853,E2 -17572.853} C_VEL
LIN {X 0,Y 287.679,Z 410.333,A -85,B 0,C 180,E1 -17574.964,E2 -17574.964} C_VEL
LIN {X 0,Y 290.594,Z 398.482,A -85,B 0,C 180,E1 -17577.161,E2 -17577.161} C_VEL
LIN {X 0,Y 293.632,Z 386.195,A -85,B 0,C 180,E1 -17578.992,E2 -17578.992} C_VEL
LIN {X 0,Y 295.979,Z 375.515,A -85,B 0,C 180,E1 -17580.304,E2 -17580.304} C_VEL
LIN {X 0,Y 298.463,Z 362.38,A -85,B 0,C 180,E1 -17581.646,E2 -17581.646} C_VEL
LIN {X 0,Y 300.527,Z 349.077,A -85,B 0,C 180,E1 -17582.738,E2 -17582.738} C_VEL
LIN {X 0,Y 302.358,Z 334.449,A -85,B 0,C 180,E1 -17583.657,E2 -17583.657} C_VEL
LIN {X 0,Y 303.802,Z 319.43,A -85,B 0,C 180,E1 -17584.325,E2 -17584.325} C_VEL
LIN {X 0,Y 304.772,Z 302.446,A -85,B 0,C 180,E1 -17584.801,E2 -17584.801} C_VEL
LIN {X 0,Y 308.614,Z 208.353,A -85,B 0,C 180,E1 -17586.949,E2 -17586.949} C_VEL
LIN {X 0,Y 301.747,Z 193.272,A -85,B 0,C 180,E1 -17588.39,E2 -17588.39} C_VEL
LIN {X 0,Y 294.258,Z 178.77,A -85,B 0,C 180,E1 -17590.015,E2 -17590.015} C_VEL
LIN {X 0,Y 288.954,Z 169.934,A -85,B 0,C 180,E1 -17591.195,E2 -17591.195} C_VEL
LIN {X 0,Y 282.423,Z 160.199,A -85,B 0,C 180,E1 -17592.703,E2 -17592.703} C_VEL
LIN {X 0,Y 280.222,Z 156.756,A -85,B 0,C 180,E1 -17593.241,E2 -17593.241} C_VEL
LIN {X 0,Y 279.984,Z 156.375,A -85,B 0,C 180,E1 -17593.301,E2 -17593.301} C_VEL
LIN {X 0,Y 276.693,Z 154.162,A -85,B 0,C 180,E1 -17594.082,E2 -17594.082} C_VEL
LIN {X 0,Y 273.535,Z 153.011,A -85,B 0,C 180,E1 -17594.994,E2 -17594.994} C_VEL
LIN {X 0,Y 271.132,Z 152.542,A -85,B 0,C 180,E1 -17596.022,E2 -17596.022} C_VEL
LIN {X 0,Y 270.162,Z 152.442,A -85,B 0,C 180,E1 -17597.004,E2 -17597.004} C_VEL
LIN {X 0,Y 270.145,Z 152.44,A -85,B 0,C 180,E1 -17597.147,E2 -17597.147} C_VEL
LIN {X 0,Y 270.154,Z 152.441,A -85,B 0,C 180,E1 -17601.365,E2 -17601.365} C_VEL
LIN {X 0,Y 270.199,Z 152.452,A -85,B 0,C 180,E1 -17605.094,E2 -17605.094} C_VEL
LIN {X 0,Y 270.172,Z 152.424,A -85,B 0,C 180,E1 -17609.141,E2 -17609.141} C_VEL
LIN {X 0,Y 270.19,Z 152.455,A -85,B 0,C 180,E1 -17612.176,E2 -17612.176} C_VEL
LIN {X 0,Y 270.186,Z 152.454,A -85,B 0,C 180,E1 -17615.563,E2 -17615.563} C_VEL
LIN {X 0,Y 270.222,Z 152.45,A -85,B 0,C 180,E1 -17620.238,E2 -17620.238} C_VEL
LIN {X 0,Y 270.364,Z 152.43,A -85,B 0,C 180,E1 -17624.933,E2 -17624.933} C_VEL
LIN {X 0,Y 270.412,Z 152.421,A -85,B 0,C 180,E1 -17629.518,E2 -17629.518} C_VEL
LIN {X 0,Y 270.564,Z 152.408,A -85,B 0,C 180,E1 -17632.537,E2 -17632.537} C_VEL
LIN {X 0,Y 270.777,Z 152.379,A -85,B 0,C 180,E1 -17638.513,E2 -17638.513} C_VEL
LIN {X 0,Y 270.78,Z 152.376,A -85,B 0,C 180,E1 -17641.487,E2 -17641.487} C_VEL
LIN {X 0,Y 270.565,Z 152.408,A -85,B 0,C 180,E1 -17647.462,E2 -17647.462} C_VEL
LIN {X 0,Y 270.412,Z 152.423,A -85,B 0,C 180,E1 -17650.482,E2 -17650.482} C_VEL
LIN {X 0,Y 270.379,Z 152.428,A -85,B 0,C 180,E1 -17655.066,E2 -17655.066} C_VEL
LIN {X 0,Y 270.292,Z 152.444,A -85,B 0,C 180,E1 -17659.756,E2 -17659.756} C_VEL
LIN {X 0,Y 270.229,Z 152.453,A -85,B 0,C 180,E1 -17664.59,E2 -17664.59} C_VEL
LIN {X 0,Y 270.21,Z 152.452,A -85,B 0,C 180,E1 -17667.915,E2 -17667.915} C_VEL
LIN {X 0,Y 270.175,Z 152.456,A -85,B 0,C 180,E1 -17671.349,E2 -17671.349} C_VEL
LIN {X 0,Y 270.203,Z 152.449,A -85,B 0,C 180,E1 -17674.905,E2 -17674.905} C_VEL
LIN {X 0,Y 270.198,Z 152.453,A -85,B 0,C 180,E1 -17678.71,E2 -17678.71} C_VEL
LIN {X 0,Y 270.194,Z 152.606,A -85,B 0,C 180,E1 -17681.721,E2 -17681.721} C_VEL
LIN {X 0,Y 272.845,Z 160.826,A -85,B 0,C 180,E1 -17685.074,E2 -17685.074} C_VEL
LIN {X 0,Y 275.71,Z 165.469,A -85,B 0,C 180,E1 -17685.826,E2 -17685.826} C_VEL
LIN {X 0,Y 284.465,Z 180.37,A -85,B 0,C 180,E1 -17688.002,E2 -17688.002} C_VEL
LIN {X 0,Y 293.086,Z 197.118,A -85,B 0,C 180,E1 -17690.018,E2 -17690.018} C_VEL
LIN {X 0,Y 300.871,Z 214.525,A -85,B 0,C 180,E1 -17691.761,E2 -17691.761} C_VEL
LIN {X 0,Y 301.873,Z 217.299,A -85,B 0,C 180,E1 -17691.992,E2 -17691.992} C_VEL
LIN {X 0,Y 302.478,Z 222.294,A -85,B 0,C 180,E1 -17692.228,E2 -17692.228} C_VEL
LIN {X 0,Y 297.896,Z 327.612,A -85,B 0,C 180,E1 -17694.689,E2 -17694.689} C_VEL
LIN {X 0,Y 296.494,Z 343.007,A -85,B 0,C 180,E1 -17695.275,E2 -17695.275} C_VEL
LIN {X 0,Y 294.478,Z 357.902,A -85,B 0,C 180,E1 -17696.091,E2 -17696.091} C_VEL
LIN {X 0,Y 292.336,Z 370.877,A -85,B 0,C 180,E1 -17697.049,E2 -17697.049} C_VEL
LIN {X 0,Y 289.637,Z 385.045,A -85,B 0,C 180,E1 -17698.388,E2 -17698.388} C_VEL
LIN {X 0,Y 286.772,Z 397.465,A -85,B 0,C 180,E1 -17699.841,E2 -17699.841} C_VEL
LIN {X 0,Y 283.536,Z 410.335,A -85,B 0,C 180,E1 -17701.702,E2 -17701.702} C_VEL
LIN {X 0,Y 280.643,Z 421.115,A -85,B 0,C 180,E1 -17703.608,E2 -17703.608} C_VEL
LIN {X 0,Y 277.824,Z 431.561,A -85,B 0,C 180,E1 -17705.851,E2 -17705.851} C_VEL
LIN {X 0,Y 275.187,Z 440.867,A -85,B 0,C 180,E1 -17708.265,E2 -17708.265} C_VEL
LIN {X 0,Y 272.839,Z 449.022,A -85,B 0,C 180,E1 -17710.827,E2 -17710.827} C_VEL
LIN {X 0,Y 270.955,Z 456.362,A -85,B 0,C 180,E1 -17713.678,E2 -17713.678} C_VEL
LIN {X 0,Y 269.674,Z 462.013,A -85,B 0,C 180,E1 -17716.435,E2 -17716.435} C_VEL
LIN {X 0,Y 268.7,Z 466.842,A -85,B 0,C 180,E1 -17719.45,E2 -17719.45} C_VEL
LIN {X 0,Y 268.237,Z 470.386,A -85,B 0,C 180,E1 -17722.472,E2 -17722.472} C_VEL
LIN {X 0,Y 268.104,Z 472.72,A -85,B 0,C 180,E1 -17725.489,E2 -17725.489} C_VEL
LIN {X 0,Y 268.181,Z 473.895,A -85,B 0,C 180,E1 -17728.498,E2 -17728.498} C_VEL
LIN {X 0,Y 268.181,Z 473.891,A -85,B 0,C 180,E1 -17731.502,E2 -17731.502} C_VEL
LIN {X 0,Y 268.106,Z 472.7,A -85,B 0,C 180,E1 -17734.51,E2 -17734.51} C_VEL
LIN {X 0,Y 268.237,Z 470.353,A -85,B 0,C 180,E1 -17737.528,E2 -17737.528} C_VEL
LIN {X 0,Y 268.699,Z 466.801,A -85,B 0,C 180,E1 -17740.55,E2 -17740.55} C_VEL
LIN {X 0,Y 269.663,Z 461.96,A -85,B 0,C 180,E1 -17743.566,E2 -17743.566} C_VEL
LIN {X 0,Y 271.002,Z 455.694,A -85,B 0,C 180,E1 -17746.575,E2 -17746.575} C_VEL
LIN {X 0,Y 273.137,Z 447.841,A -85,B 0,C 180,E1 -17749.542,E2 -17749.542} C_VEL
LIN {X 0,Y 275.543,Z 439.496,A -85,B 0,C 180,E1 -17752.099,E2 -17752.099} C_VEL
LIN {X 0,Y 278.235,Z 429.622,A -85,B 0,C 180,E1 -17754.587,E2 -17754.587} C_VEL
LIN {X 0,Y 281.121,Z 419.173,A -85,B 0,C 180,E1 -17756.744,E2 -17756.744} C_VEL
LIN {X 0,Y 284.374,Z 406.936,A -85,B 0,C 180,E1 -17758.811,E2 -17758.811} C_VEL
LIN {X 0,Y 287.742,Z 393.313,A -85,B 0,C 180,E1 -17760.655,E2 -17760.655} C_VEL
LIN {X 0,Y 290.629,Z 379.651,A -85,B 0,C 180,E1 -17762.141,E2 -17762.141} C_VEL
LIN {X 0,Y 293.17,Z 365.498,A -85,B 0,C 180,E1 -17763.358,E2 -17763.358} C_VEL
LIN {X 0,Y 295.527,Z 350.18,A -85,B 0,C 180,E1 -17764.337,E2 -17764.337} C_VEL
LIN {X 0,Y 297.224,Z 334.883,A -85,B 0,C 180,E1 -17765.04,E2 -17765.04} C_VEL
LIN {X 0,Y 298.294,Z 318.761,A -85,B 0,C 180,E1 -17765.515,E2 -17765.515} C_VEL
LIN {X 0,Y 301.741,Z 236.902,A -85,B 0,C 180,E1 -17767.413,E2 -17767.413} C_VEL
LIN {X 0,Y 302.368,Z 220.95,A -85,B 0,C 180,E1 -17767.79,E2 -17767.79} C_VEL
LIN {X 0,Y 301.511,Z 216.187,A -85,B 0,C 180,E1 -17768.055,E2 -17768.055} C_VEL
LIN {X 0,Y 293.864,Z 198.813,A -85,B 0,C 180,E1 -17769.76,E2 -17769.76} C_VEL
LIN {X 0,Y 286.369,Z 184.042,A -85,B 0,C 180,E1 -17771.49,E2 -17771.49} C_VEL
LIN {X 0,Y 280.28,Z 173.26,A -85,B 0,C 180,E1 -17772.96,E2 -17772.96} C_VEL
LIN {X 0,Y 275.109,Z 164.685,A -85,B 0,C 180,E1 -17774.267,E2 -17774.267} C_VEL
LIN {X 0,Y 272.686,Z 160.495,A -85,B 0,C 180,E1 -17774.954,E2 -17774.954} C_VEL
LIN {X 0,Y 270.149,Z 152.456,A -85,B 0,C 180,E1 -17778.322,E2 -17778.322} C_VEL
LIN {X 0,Y 270.207,Z 152.444,A -85,B 0,C 180,E1 -17781.374,E2 -17781.374} C_VEL
LIN {X 0,Y 270.202,Z 152.447,A -85,B 0,C 180,E1 -17785.095,E2 -17785.095} C_VEL
LIN {X 0,Y 270.201,Z 152.447,A -85,B 0,C 180,E1 -17789.131,E2 -17789.131} C_VEL
LIN {X 0,Y 270.266,Z 152.442,A -85,B 0,C 180,E1 -17792.146,E2 -17792.146} C_VEL
LIN {X 0,Y 270.278,Z 152.44,A -85,B 0,C 180,E1 -17795.519,E2 -17795.519} C_VEL
LIN {X 0,Y 270.303,Z 152.431,A -85,B 0,C 180,E1 -17800.245,E2 -17800.245} C_VEL
LIN {X 0,Y 270.405,Z 152.425,A -85,B 0,C 180,E1 -17804.936,E2 -17804.936} C_VEL
LIN {X 0,Y 270.412,Z 152.426,A -85,B 0,C 180,E1 -17809.518,E2 -17809.518} C_VEL
LIN {X 0,Y 270.565,Z 152.4,A -85,B 0,C 180,E1 -17812.538,E2 -17812.538} C_VEL
LIN {X 0,Y 270.779,Z 152.38,A -85,B 0,C 180,E1 -17818.513,E2 -17818.513} C_VEL
LIN {X 0,Y 270.778,Z 152.378,A -85,B 0,C 180,E1 -17821.487,E2 -17821.487} C_VEL
LIN {X 0,Y 270.564,Z 152.407,A -85,B 0,C 180,E1 -17827.463,E2 -17827.463} C_VEL
LIN {X 0,Y 270.41,Z 152.426,A -85,B 0,C 180,E1 -17830.482,E2 -17830.482} C_VEL
LIN {X 0,Y 270.353,Z 152.434,A -85,B 0,C 180,E1 -17835.068,E2 -17835.068} C_VEL
LIN {X 0,Y 270.261,Z 152.444,A -85,B 0,C 180,E1 -17839.759,E2 -17839.759} C_VEL
LIN {X 0,Y 270.225,Z 152.433,A -85,B 0,C 180,E1 -17844.59,E2 -17844.59} C_VEL
LIN {X 0,Y 270.199,Z 152.43,A -85,B 0,C 180,E1 -17847.917,E2 -17847.917} C_VEL
LIN {X 0,Y 270.175,Z 152.45,A -85,B 0,C 180,E1 -17851.35,E2 -17851.35} C_VEL
LIN {X 0,Y 270.199,Z 152.446,A -85,B 0,C 180,E1 -17854.906,E2 -17854.906} C_VEL
LIN {X 0,Y 270.199,Z 152.451,A -85,B 0,C 180,E1 -17858.71,E2 -17858.71} C_VEL
LIN {X 0,Y 270.149,Z 152.456,A -85,B 0,C 180,E1 -17863.245,E2 -17863.245} C_VEL
LIN {X 0,Y 270.156,Z 152.574,A -85,B 0,C 180,E1 -17864.698,E2 -17864.698} C_VEL
LIN {X 0,Y 271.121,Z 155.292,A -85,B 0,C 180,E1 -17865.006,E2 -17865.006} C_VEL
LIN {X 0,Y 273.353,Z 157.86,A -85,B 0,C 180,E1 -17865.568,E2 -17865.568} C_VEL
LIN {X 0,Y 275.517,Z 161.2,A -85,B 0,C 180,E1 -17866.13,E2 -17866.13} C_VEL
LIN {X 0,Y 282.686,Z 171.728,A -85,B 0,C 180,E1 -17867.877,E2 -17867.877} C_VEL
LIN {X 0,Y 288.366,Z 180.804,A -85,B 0,C 180,E1 -17869.191,E2 -17869.191} C_VEL
LIN {X 0,Y 296.419,Z 196.402,A -85,B 0,C 180,E1 -17871.012,E2 -17871.012} C_VEL
LIN {X 0,Y 302.747,Z 210.231,A -85,B 0,C 180,E1 -17872.39,E2 -17872.39} C_VEL
LIN {X 0,Y 299.468,Z 287.511,A -85,B 0,C 180,E1 -17874.18,E2 -17874.18} C_VEL
LIN {X 0,Y 298.157,Z 315.681,A -85,B 0,C 180,E1 -17874.88,E2 -17874.88} C_VEL
LIN {X 0,Y 296.92,Z 330.231,A -85,B 0,C 180,E1 -17875.469,E2 -17875.469} C_VEL
LIN {X 0,Y 295.295,Z 343.95,A -85,B 0,C 180,E1 -17876.26,E2 -17876.26} C_VEL
LIN {X 0,Y 293.177,Z 358.086,A -85,B 0,C 180,E1 -17877.339,E2 -17877.339} C_VEL
LIN {X 0,Y 290.572,Z 371.847,A -85,B 0,C 180,E1 -17878.667,E2 -17878.667} C_VEL
LIN {X 0,Y 287.822,Z 384.322,A -85,B 0,C 180,E1 -17880.164,E2 -17880.164} C_VEL
LIN {X 0,Y 284.713,Z 396.958,A -85,B 0,C 180,E1 -17882.03,E2 -17882.03} C_VEL
LIN {X 0,Y 281.633,Z 408.483,A -85,B 0,C 180,E1 -17884.122,E2 -17884.122} C_VEL
LIN {X 0,Y 278.939,Z 418.048,A -85,B 0,C 180,E1 -17886.226,E2 -17886.226} C_VEL
LIN {X 0,Y 276.234,Z 427.488,A -85,B 0,C 180,E1 -17888.743,E2 -17888.743} C_VEL
LIN {X 0,Y 273.526,Z 436.347,A -85,B 0,C 180,E1 -17891.654,E2 -17891.654} C_VEL
LIN {X 0,Y 271.86,Z 442.674,A -85,B 0,C 180,E1 -17894.25,E2 -17894.25} C_VEL
LIN {X 0,Y 270.239,Z 448.487,A -85,B 0,C 180,E1 -17897.229,E2 -17897.229} C_VEL
LIN {X 0,Y 269.467,Z 451.924,A -85,B 0,C 180,E1 -17899.481,E2 -17899.481} C_VEL
LIN {X 0,Y 268.781,Z 455.403,A -85,B 0,C 180,E1 -17902.488,E2 -17902.488} C_VEL
LIN {X 0,Y 268.38,Z 457.702,A -85,B 0,C 180,E1 -17905.494,E2 -17905.494} C_VEL
LIN {X 0,Y 268.225,Z 458.873,A -85,B 0,C 180,E1 -17908.499,E2 -17908.499} C_VEL
LIN {X 0,Y 268.225,Z 458.886,A -85,B 0,C 180,E1 -17911.502,E2 -17911.502} C_VEL
LIN {X 0,Y 268.379,Z 457.769,A -85,B 0,C 180,E1 -17914.506,E2 -17914.506} C_VEL
LIN {X 0,Y 268.776,Z 455.522,A -85,B 0,C 180,E1 -17917.513,E2 -17917.513} C_VEL
LIN {X 0,Y 269.445,Z 452.092,A -85,B 0,C 180,E1 -17920.52,E2 -17920.52} C_VEL
LIN {X 0,Y 270.532,Z 447.392,A -85,B 0,C 180,E1 -17923.521,E2 -17923.521} C_VEL
LIN {X 0,Y 272.22,Z 441.295,A -85,B 0,C 180,E1 -17926.499,E2 -17926.499} C_VEL
LIN {X 0,Y 274.398,Z 433.616,A -85,B 0,C 180,E1 -17929.449,E2 -17929.449} C_VEL
LIN {X 0,Y 276.856,Z 425.422,A -85,B 0,C 180,E1 -17931.989,E2 -17931.989} C_VEL
LIN {X 0,Y 279.813,Z 415.545,A -85,B 0,C 180,E1 -17934.483,E2 -17934.483} C_VEL
LIN {X 0,Y 282.545,Z 405.421,A -85,B 0,C 180,E1 -17936.598,E2 -17936.598} C_VEL
LIN {X 0,Y 285.148,Z 395.486,A -85,B 0,C 180,E1 -17938.324,E2 -17938.324} C_VEL
LIN {X 0,Y 287.963,Z 383.828,A -85,B 0,C 180,E1 -17940.022,E2 -17940.022} C_VEL
LIN {X 0,Y 290.783,Z 371.251,A -85,B 0,C 180,E1 -17941.511,E2 -17941.511} C_VEL
LIN {X 0,Y 293.311,Z 357.17,A -85,B 0,C 180,E1 -17942.866,E2 -17942.866} C_VEL
LIN {X 0,Y 295.39,Z 343.463,A -85,B 0,C 180,E1 -17943.892,E2 -17943.892} C_VEL
LIN {X 0,Y 297.16,Z 328.318,A -85,B 0,C 180,E1 -17944.739,E2 -17944.739} C_VEL
LIN {X 0,Y 298.457,Z 313.799,A -85,B 0,C 180,E1 -17945.286,E2 -17945.286} C_VEL
LIN {X 0,Y 301.923,Z 232.241,A -85,B 0,C 180,E1 -17947.212,E2 -17947.212} C_VEL
LIN {X 0,Y 302.859,Z 210.419,A -85,B 0,C 180,E1 -17947.717,E2 -17947.717} C_VEL
LIN {X 0,Y 295.846,Z 195.157,A -85,B 0,C 180,E1 -17949.25,E2 -17949.25} C_VEL
LIN {X 0,Y 289.14,Z 182.217,A -85,B 0,C 180,E1 -17950.766,E2 -17950.766} C_VEL
LIN {X 0,Y 283.477,Z 172.872,A -85,B 0,C 180,E1 -17952.079,E2 -17952.079} C_VEL
LIN {X 0,Y 278.138,Z 164.986,A -85,B 0,C 180,E1 -17953.361,E2 -17953.361} C_VEL
LIN {X 0,Y 275.536,Z 161.194,A -85,B 0,C 180,E1 -17954.012,E2 -17954.012} C_VEL
LIN {X 0,Y 273.388,Z 157.921,A -85,B 0,C 180,E1 -17954.57,E2 -17954.57} C_VEL
LIN {X 0,Y 270.866,Z 154.825,A -85,B 0,C 180,E1 -17955.215,E2 -17955.215} C_VEL
LIN {X 0,Y 270.129,Z 152.463,A -85,B 0,C 180,E1 -17955.469,E2 -17955.469} C_VEL
LIN {X 0,Y 270.145,Z 152.44,A -85,B 0,C 180,E1 -17957.147,E2 -17957.147} C_VEL
LIN {X 0,Y 269.492,Z 152.525,A -85,B 0,C 180,E1 -17958.391,E2 -17958.391} C_VEL
LIN {X 0,Y 266.653,Z 152.893,A -85,B 0,C 180,E1 -17960.419,E2 -17960.419} C_VEL
LIN {X 0,Y 264.244,Z 153.178,A -85,B 0,C 180,E1 -17962.067,E2 -17962.067} C_VEL
LIN {X 0,Y 263.224,Z 153.298,A -85,B 0,C 180,E1 -17963.345,E2 -17963.345} C_VEL
LIN {X 0,Y 263.149,Z 153.31,A -85,B 0,C 180,E1 -17963.777,E2 -17963.777} C_VEL
LIN {X 0,Y 263.127,Z 153.305,A -85,B 0,C 180,E1 -17967.711,E2 -17967.711} C_VEL
LIN {X 0,Y 263.138,Z 153.332,A -85,B 0,C 180,E1 -17971.809,E2 -17971.809} C_VEL
LIN {X 0,Y 263.119,Z 153.333,A -85,B 0,C 180,E1 -17976.381,E2 -17976.381} C_VEL
LIN {X 0,Y 263.209,Z 153.324,A -85,B 0,C 180,E1 -17979.689,E2 -17979.689} C_VEL
LIN {X 0,Y 263.306,Z 153.31,A -85,B 0,C 180,E1 -17984.519,E2 -17984.519} C_VEL
LIN {X 0,Y 263.352,Z 153.304,A -85,B 0,C 180,E1 -17989.233,E2 -17989.233} C_VEL
LIN {X 0,Y 263.528,Z 153.282,A -85,B 0,C 180,E1 -17992.337,E2 -17992.337} C_VEL
LIN {X 0,Y 263.74,Z 153.255,A -85,B 0,C 180,E1 -17998.473,E2 -17998.473} C_VEL
LIN {X 0,Y 263.745,Z 153.252,A -85,B 0,C 180,E1 -18001.527,E2 -18001.527} C_VEL
LIN {X 0,Y 263.529,Z 153.283,A -85,B 0,C 180,E1 -18007.663,E2 -18007.663} C_VEL
LIN {X 0,Y 263.355,Z 153.304,A -85,B 0,C 180,E1 -18010.766,E2 -18010.766} C_VEL
LIN {X 0,Y 263.326,Z 153.311,A -85,B 0,C 180,E1 -18015.479,E2 -18015.479} C_VEL
LIN {X 0,Y 263.258,Z 153.321,A -85,B 0,C 180,E1 -18020.307,E2 -18020.307} C_VEL
LIN {X 0,Y 263.174,Z 153.326,A -85,B 0,C 180,E1 -18025.295,E2 -18025.295} C_VEL
LIN {X 0,Y 263.14,Z 153.333,A -85,B 0,C 180,E1 -18028.734,E2 -18028.734} C_VEL
LIN {X 0,Y 263.129,Z 153.334,A -85,B 0,C 180,E1 -18032.289,E2 -18032.289} C_VEL
LIN {X 0,Y 263.184,Z 153.319,A -85,B 0,C 180,E1 -18036.763,E2 -18036.763} C_VEL
LIN {X 0,Y 263.134,Z 153.371,A -85,B 0,C 180,E1 -18040.367,E2 -18040.367} C_VEL
LIN {X 0,Y 265.408,Z 160.432,A -85,B 0,C 180,E1 -18043.444,E2 -18043.444} C_VEL
LIN {X 0,Y 268.41,Z 165.259,A -85,B 0,C 180,E1 -18044.294,E2 -18044.294} C_VEL
LIN {X 0,Y 275.328,Z 176.655,A -85,B 0,C 180,E1 -18046.146,E2 -18046.146} C_VEL
LIN {X 0,Y 282.369,Z 189.296,A -85,B 0,C 180,E1 -18047.92,E2 -18047.92} C_VEL
LIN {X 0,Y 289.975,Z 204.732,A -85,B 0,C 180,E1 -18049.746,E2 -18049.746} C_VEL
LIN {X 0,Y 296.498,Z 219.949,A -85,B 0,C 180,E1 -18051.261,E2 -18051.261} C_VEL
LIN {X 0,Y 296.828,Z 223.757,A -85,B 0,C 180,E1 -18051.427,E2 -18051.427} C_VEL
LIN {X 0,Y 292.142,Z 327.43,A -85,B 0,C 180,E1 -18053.886,E2 -18053.886} C_VEL
LIN {X 0,Y 290.696,Z 342.819,A -85,B 0,C 180,E1 -18054.479,E2 -18054.479} C_VEL
LIN {X 0,Y 288.606,Z 357.711,A -85,B 0,C 180,E1 -18055.304,E2 -18055.304} C_VEL
LIN {X 0,Y 286.278,Z 371.275,A -85,B 0,C 180,E1 -18056.323,E2 -18056.323} C_VEL
LIN {X 0,Y 283.471,Z 385.438,A -85,B 0,C 180,E1 -18057.696,E2 -18057.696} C_VEL
LIN {X 0,Y 280.304,Z 398.564,A -85,B 0,C 180,E1 -18059.279,E2 -18059.279} C_VEL
LIN {X 0,Y 276.983,Z 411.212,A -85,B 0,C 180,E1 -18061.177,E2 -18061.177} C_VEL
LIN {X 0,Y 273.728,Z 422.708,A -85,B 0,C 180,E1 -18063.3,E2 -18063.3} C_VEL
LIN {X 0,Y 270.991,Z 432.393,A -85,B 0,C 180,E1 -18065.484,E2 -18065.484} C_VEL
LIN {X 0,Y 268.139,Z 441.907,A -85,B 0,C 180,E1 -18068.068,E2 -18068.068} C_VEL
LIN {X 0,Y 265.784,Z 449.839,A -85,B 0,C 180,E1 -18070.699,E2 -18070.699} C_VEL
LIN {X 0,Y 263.776,Z 457.253,A -85,B 0,C 180,E1 -18073.754,E2 -18073.754} C_VEL
LIN {X 0,Y 262.406,Z 463.14,A -85,B 0,C 180,E1 -18076.841,E2 -18076.841} C_VEL
LIN {X 0,Y 261.661,Z 466.642,A -85,B 0,C 180,E1 -18079.163,E2 -18079.163} C_VEL
LIN {X 0,Y 261.15,Z 470.186,A -85,B 0,C 180,E1 -18082.267,E2 -18082.267} C_VEL
LIN {X 0,Y 261.017,Z 472.521,A -85,B 0,C 180,E1 -18085.367,E2 -18085.367} C_VEL
LIN {X 0,Y 261.108,Z 473.697,A -85,B 0,C 180,E1 -18088.458,E2 -18088.458} C_VEL
LIN {X 0,Y 261.108,Z 473.693,A -85,B 0,C 180,E1 -18091.542,E2 -18091.542} C_VEL
LIN {X 0,Y 261.084,Z 472.233,A -85,B 0,C 180,E1 -18095.137,E2 -18095.137} C_VEL
LIN {X 0,Y 261.15,Z 470.152,A -85,B 0,C 180,E1 -18097.733,E2 -18097.733} C_VEL
LIN {X 0,Y 261.659,Z 466.6,A -85,B 0,C 180,E1 -18100.837,E2 -18100.837} C_VEL
LIN {X 0,Y 262.684,Z 461.758,A -85,B 0,C 180,E1 -18103.933,E2 -18103.933} C_VEL
LIN {X 0,Y 264.155,Z 455.492,A -85,B 0,C 180,E1 -18107.017,E2 -18107.017} C_VEL
LIN {X 0,Y 266.373,Z 447.638,A -85,B 0,C 180,E1 -18110.059,E2 -18110.059} C_VEL
LIN {X 0,Y 268.928,Z 439.294,A -85,B 0,C 180,E1 -18112.673,E2 -18112.673} C_VEL
LIN {X 0,Y 271.868,Z 428.997,A -85,B 0,C 180,E1 -18115.309,E2 -18115.309} C_VEL
LIN {X 0,Y 274.758,Z 418.971,A -85,B 0,C 180,E1 -18117.414,E2 -18117.414} C_VEL
LIN {X 0,Y 278.114,Z 406.732,A -85,B 0,C 180,E1 -18119.523,E2 -18119.523} C_VEL
LIN {X 0,Y 281.637,Z 393.109,A -85,B 0,C 180,E1 -18121.394,E2 -18121.394} C_VEL
LIN {X 0,Y 284.612,Z 379.446,A -85,B 0,C 180,E1 -18122.905,E2 -18122.905} C_VEL
LIN {X 0,Y 287.258,Z 365.291,A -85,B 0,C 180,E1 -18124.138,E2 -18124.138} C_VEL
LIN {X 0,Y 289.678,Z 349.971,A -85,B 0,C 180,E1 -18125.131,E2 -18125.131} C_VEL
LIN {X 0,Y 291.437,Z 334.671,A -85,B 0,C 180,E1 -18125.841,E2 -18125.841} C_VEL
LIN {X 0,Y 292.556,Z 318.542,A -85,B 0,C 180,E1 -18126.321,E2 -18126.321} C_VEL
LIN {X 0,Y 296.733,Z 223.652,A -85,B 0,C 180,E1 -18128.55,E2 -18128.55} C_VEL
LIN {X 0,Y 296.407,Z 219.784,A -85,B 0,C 180,E1 -18128.717,E2 -18128.717} C_VEL
LIN {X 0,Y 289.306,Z 203.252,A -85,B 0,C 180,E1 -18130.368,E2 -18130.368} C_VEL
LIN {X 0,Y 281.823,Z 188.4,A -85,B 0,C 180,E1 -18132.16,E2 -18132.16} C_VEL
LIN {X 0,Y 274.661,Z 175.485,A -85,B 0,C 180,E1 -18133.974,E2 -18133.974} C_VEL
LIN {X 0,Y 267.938,Z 164.628,A -85,B 0,C 180,E1 -18135.772,E2 -18135.772} C_VEL
LIN {X 0,Y 265.278,Z 160.147,A -85,B 0,C 180,E1 -18136.594,E2 -18136.594} C_VEL
LIN {X 0,Y 263.131,Z 153.328,A -85,B 0,C 180,E1 -18139.632,E2 -18139.632} C_VEL
LIN {X 0,Y 263.163,Z 153.32,A -85,B 0,C 180,E1 -18144.018,E2 -18144.018} C_VEL
LIN {X 0,Y 263.134,Z 153.326,A -85,B 0,C 180,E1 -18147.712,E2 -18147.712} C_VEL
LIN {X 0,Y 263.203,Z 153.323,A -85,B 0,C 180,E1 -18151.783,E2 -18151.783} C_VEL
LIN {X 0,Y 263.227,Z 153.32,A -85,B 0,C 180,E1 -18155.201,E2 -18155.201} C_VEL
LIN {X 0,Y 263.265,Z 153.308,A -85,B 0,C 180,E1 -18159.694,E2 -18159.694} C_VEL
LIN {X 0,Y 263.353,Z 153.299,A -85,B 0,C 180,E1 -18164.522,E2 -18164.522} C_VEL
LIN {X 0,Y 263.352,Z 153.307,A -85,B 0,C 180,E1 -18169.234,E2 -18169.234} C_VEL
LIN {X 0,Y 263.528,Z 153.274,A -85,B 0,C 180,E1 -18172.337,E2 -18172.337} C_VEL
LIN {X 0,Y 263.745,Z 153.257,A -85,B 0,C 180,E1 -18178.473,E2 -18178.473} C_VEL
LIN {X 0,Y 263.741,Z 153.254,A -85,B 0,C 180,E1 -18181.527,E2 -18181.527} C_VEL
LIN {X 0,Y 263.528,Z 153.281,A -85,B 0,C 180,E1 -18187.663,E2 -18187.663} C_VEL
LIN {X 0,Y 263.349,Z 153.307,A -85,B 0,C 180,E1 -18190.767,E2 -18190.767} C_VEL
LIN {X 0,Y 263.3,Z 153.313,A -85,B 0,C 180,E1 -18195.481,E2 -18195.481} C_VEL
LIN {X 0,Y 263.24,Z 153.314,A -85,B 0,C 180,E1 -18200.309,E2 -18200.309} C_VEL
LIN {X 0,Y 263.168,Z 153.301,A -85,B 0,C 180,E1 -18205.296,E2 -18205.296} C_VEL
LIN {X 0,Y 263.134,Z 153.323,A -85,B 0,C 180,E1 -18208.735,E2 -18208.735} C_VEL
LIN {X 0,Y 263.129,Z 153.332,A -85,B 0,C 180,E1 -18212.289,E2 -18212.289} C_VEL
LIN {X 0,Y 263.177,Z 153.321,A -85,B 0,C 180,E1 -18216.761,E2 -18216.761} C_VEL
LIN {X 0,Y 263.092,Z 153.33,A -85,B 0,C 180,E1 -18219.875,E2 -18219.875} C_VEL
LIN {X 0,Y 263.11,Z 153.332,A -85,B 0,C 180,E1 -18223.126,E2 -18223.126} C_VEL
LIN {X 0,Y 264.043,Z 156.102,A -85,B 0,C 180,E1 -18223.468,E2 -18223.468} C_VEL
LIN {X 0,Y 266.461,Z 158.925,A -85,B 0,C 180,E1 -18224.125,E2 -18224.125} C_VEL
LIN {X 0,Y 268.526,Z 162.089,A -85,B 0,C 180,E1 -18224.7,E2 -18224.7} C_VEL
LIN {X 0,Y 269.83,Z 163.756,A -85,B 0,C 180,E1 -18225.043,E2 -18225.043} C_VEL
LIN {X 0,Y 278.689,Z 176.843,A -85,B 0,C 180,E1 -18227.3,E2 -18227.3} C_VEL
LIN {X 0,Y 284.299,Z 186.081,A -85,B 0,C 180,E1 -18228.649,E2 -18228.649} C_VEL
LIN {X 0,Y 291.974,Z 201.192,A -85,B 0,C 180,E1 -18230.447,E2 -18230.447} C_VEL
LIN {X 0,Y 297.144,Z 212.6,A -85,B 0,C 180,E1 -18231.618,E2 -18231.618} C_VEL
LIN {X 0,Y 292.489,Z 314.745,A -85,B 0,C 180,E1 -18234.042,E2 -18234.042} C_VEL
LIN {X 0,Y 291.155,Z 329.924,A -85,B 0,C 180,E1 -18234.65,E2 -18234.65} C_VEL
LIN {X 0,Y 289.347,Z 344.67,A -85,B 0,C 180,E1 -18235.511,E2 -18235.511} C_VEL
LIN {X 0,Y 287.153,Z 358.73,A -85,B 0,C 180,E1 -18236.611,E2 -18236.611} C_VEL
LIN {X 0,Y 284.207,Z 373.605,A -85,B 0,C 180,E1 -18238.091,E2 -18238.091} C_VEL
LIN {X 0,Y 281.401,Z 385.811,A -85,B 0,C 180,E1 -18239.619,E2 -18239.619} C_VEL
LIN {X 0,Y 278.166,Z 398.225,A -85,B 0,C 180,E1 -18241.518,E2 -18241.518} C_VEL
LIN {X 0,Y 275.106,Z 409.185,A -85,B 0,C 180,E1 -18243.576,E2 -18243.576} C_VEL
LIN {X 0,Y 272.432,Z 418.25,A -85,B 0,C 180,E1 -18245.622,E2 -18245.622} C_VEL
LIN {X 0,Y 269.578,Z 427.691,A -85,B 0,C 180,E1 -18248.192,E2 -18248.192} C_VEL
LIN {X 0,Y 267.064,Z 435.549,A -85,B 0,C 180,E1 -18250.795,E2 -18250.795} C_VEL
LIN {X 0,Y 265.399,Z 441.209,A -85,B 0,C 180,E1 -18253.065,E2 -18253.065} C_VEL
LIN {X 0,Y 264.093,Z 445.96,A -85,B 0,C 180,E1 -18255.356,E2 -18255.356} C_VEL
LIN {X 0,Y 262.714,Z 451.074,A -85,B 0,C 180,E1 -18258.426,E2 -18258.426} C_VEL
LIN {X 0,Y 262.057,Z 454.016,A -85,B 0,C 180,E1 -18260.74,E2 -18260.74} C_VEL
LIN {X 0,Y 261.44,Z 456.896,A -85,B 0,C 180,E1 -18263.827,E2 -18263.827} C_VEL
LIN {X 0,Y 261.22,Z 458.624,A -85,B 0,C 180,E1 -18266.916,E2 -18266.916} C_VEL
LIN {X 0,Y 261.133,Z 459.227,A -85,B 0,C 180,E1 -18270,E2 -18270} C_VEL
LIN {X 0,Y 261.22,Z 458.664,A -85,B 0,C 180,E1 -18273.085,E2 -18273.085} C_VEL
LIN {X 0,Y 261.44,Z 456.989,A -85,B 0,C 180,E1 -18276.173,E2 -18276.173} C_VEL
LIN {X 0,Y 262.017,Z 454.159,A -85,B 0,C 180,E1 -18279.261,E2 -18279.261} C_VEL
LIN {X 0,Y 262.959,Z 450.106,A -85,B 0,C 180,E1 -18282.346,E2 -18282.346} C_VEL
LIN {X 0,Y 264.504,Z 444.724,A -85,B 0,C 180,E1 -18285.409,E2 -18285.409} C_VEL
LIN {X 0,Y 266.473,Z 437.866,A -85,B 0,C 180,E1 -18288.451,E2 -18288.451} C_VEL
LIN {X 0,Y 268.732,Z 430.488,A -85,B 0,C 180,E1 -18291.076,E2 -18291.076} C_VEL
LIN {X 0,Y 271.504,Z 421.59,A -85,B 0,C 180,E1 -18293.655,E2 -18293.655} C_VEL
LIN {X 0,Y 274.667,Z 411.227,A -85,B 0,C 180,E1 -18296.108,E2 -18296.108} C_VEL
LIN {X 0,Y 277.737,Z 399.862,A -85,B 0,C 180,E1 -18298.324,E2 -18298.324} C_VEL
LIN {X 0,Y 280.981,Z 387.767,A -85,B 0,C 180,E1 -18300.224,E2 -18300.224} C_VEL
LIN {X 0,Y 283.809,Z 375.903,A -85,B 0,C 180,E1 -18301.75,E2 -18301.75} C_VEL
LIN {X 0,Y 286.55,Z 362.168,A -85,B 0,C 180,E1 -18303.198,E2 -18303.198} C_VEL
LIN {X 0,Y 288.85,Z 348.332,A -85,B 0,C 180,E1 -18304.345,E2 -18304.345} C_VEL
LIN {X 0,Y 290.862,Z 333.303,A -85,B 0,C 180,E1 -18305.285,E2 -18305.285} C_VEL
LIN {X 0,Y 292.212,Z 319.796,A -85,B 0,C 180,E1 -18305.891,E2 -18305.891} C_VEL
LIN {X 0,Y 293.247,Z 302.795,A -85,B 0,C 180,E1 -18306.382,E2 -18306.382} C_VEL
LIN {X 0,Y 297.202,Z 212.499,A -85,B 0,C 180,E1 -18308.507,E2 -18308.507} C_VEL
LIN {X 0,Y 289.631,Z 196.273,A -85,B 0,C 180,E1 -18310.232,E2 -18310.232} C_VEL
LIN {X 0,Y 282.671,Z 183.11,A -85,B 0,C 180,E1 -18311.884,E2 -18311.884} C_VEL
LIN {X 0,Y 274.645,Z 170.744,A -85,B 0,C 180,E1 -18313.852,E2 -18313.852} C_VEL
LIN {X 0,Y 268.847,Z 162.437,A -85,B 0,C 180,E1 -18315.368,E2 -18315.368} C_VEL
LIN {X 0,Y 266.59,Z 159.187,A -85,B 0,C 180,E1 -18315.988,E2 -18315.988} C_VEL
LIN {X 0,Y 265.866,Z 158.139,A -85,B 0,C 180,E1 -18316.191,E2 -18316.191} C_VEL
LIN {X 0,Y 263.871,Z 155.753,A -85,B 0,C 180,E1 -18316.74,E2 -18316.74} C_VEL
LIN {X 0,Y 263.1,Z 153.318,A -85,B 0,C 180,E1 -18317.017,E2 -18317.017} C_VEL
LIN {X 0,Y 263.091,Z 153.33,A -85,B 0,C 180,E1 -18320.777,E2 -18320.777} C_VEL
LIN {X 0,Y 263.149,Z 153.31,A -85,B 0,C 180,E1 -18323.777,E2 -18323.777} C_VEL
LIN {X 0,Y 262.492,Z 153.412,A -85,B 0,C 180,E1 -18325.055,E2 -18325.055} C_VEL
LIN {X 0,Y 259.612,Z 153.75,A -85,B 0,C 180,E1 -18327.136,E2 -18327.136} C_VEL
LIN {X 0,Y 257.162,Z 154.048,A -85,B 0,C 180,E1 -18328.83,E2 -18328.83} C_VEL
LIN {X 0,Y 256.121,Z 154.182,A -85,B 0,C 180,E1 -18330.144,E2 -18330.144} C_VEL
LIN {X 0,Y 256.043,Z 154.197,A -85,B 0,C 180,E1 -18330.589,E2 -18330.589} C_VEL
LIN {X 0,Y 256.086,Z 154.206,A -85,B 0,C 180,E1 -18334.912,E2 -18334.912} C_VEL
LIN {X 0,Y 256.123,Z 154.204,A -85,B 0,C 180,E1 -18339.101,E2 -18339.101} C_VEL
LIN {X 0,Y 256.227,Z 154.195,A -85,B 0,C 180,E1 -18344.08,E2 -18344.08} C_VEL
LIN {X 0,Y 256.293,Z 154.185,A -85,B 0,C 180,E1 -18348.933,E2 -18348.933} C_VEL
LIN {X 0,Y 256.47,Z 154.158,A -85,B 0,C 180,E1 -18352.125,E2 -18352.125} C_VEL
LIN {X 0,Y 256.454,Z 154.162,A -85,B 0,C 180,E1 -18356.858,E2 -18356.858} C_VEL
LIN {X 0,Y 256.702,Z 154.132,A -85,B 0,C 180,E1 -18358.431,E2 -18358.431} C_VEL
LIN {X 0,Y 256.709,Z 154.129,A -85,B 0,C 180,E1 -18361.569,E2 -18361.569} C_VEL
LIN {X 0,Y 256.46,Z 154.163,A -85,B 0,C 180,E1 -18366.293,E2 -18366.293} C_VEL
LIN {X 0,Y 256.429,Z 154.157,A -85,B 0,C 180,E1 -18369.465,E2 -18369.465} C_VEL
LIN {X 0,Y 256.239,Z 154.183,A -85,B 0,C 180,E1 -18374.291,E2 -18374.291} C_VEL
LIN {X 0,Y 256.183,Z 154.191,A -85,B 0,C 180,E1 -18377.564,E2 -18377.564} C_VEL
LIN {X 0,Y 256.151,Z 154.202,A -85,B 0,C 180,E1 -18381.115,E2 -18381.115} C_VEL
LIN {X 0,Y 256.161,Z 154.2,A -85,B 0,C 180,E1 -18385.124,E2 -18385.124} C_VEL
LIN {X 0,Y 256.059,Z 154.214,A -85,B 0,C 180,E1 -18389.606,E2 -18389.606} C_VEL
LIN {X 0,Y 256.067,Z 154.204,A -85,B 0,C 180,E1 -18393.293,E2 -18393.293} C_VEL
LIN {X 0,Y 256.116,Z 154.199,A -85,B 0,C 180,E1 -18397.27,E2 -18397.27} C_VEL
LIN {X 0,Y 256.1,Z 154.399,A -85,B 0,C 180,E1 -18399.01,E2 -18399.01} C_VEL
LIN {X 0,Y 258.123,Z 160.272,A -85,B 0,C 180,E1 -18401.713,E2 -18401.713} C_VEL
LIN {X 0,Y 260.859,Z 164.751,A -85,B 0,C 180,E1 -18402.557,E2 -18402.557} C_VEL
LIN {X 0,Y 265.826,Z 172.576,A -85,B 0,C 180,E1 -18404.002,E2 -18404.002} C_VEL
LIN {X 0,Y 271.621,Z 182.246,A -85,B 0,C 180,E1 -18405.597,E2 -18405.597} C_VEL
LIN {X 0,Y 278.314,Z 194.558,A -85,B 0,C 180,E1 -18407.346,E2 -18407.346} C_VEL
LIN {X 0,Y 285.429,Z 209.184,A -85,B 0,C 180,E1 -18409.118,E2 -18409.118} C_VEL
LIN {X 0,Y 291.203,Z 222.987,A -85,B 0,C 180,E1 -18410.521,E2 -18410.521} C_VEL
LIN {X 0,Y 288.177,Z 292.051,A -85,B 0,C 180,E1 -18412.188,E2 -18412.188} C_VEL
LIN {X 0,Y 286.339,Z 328.466,A -85,B 0,C 180,E1 -18413.089,E2 -18413.089} C_VEL
LIN {X 0,Y 284.74,Z 344.218,A -85,B 0,C 180,E1 -18413.729,E2 -18413.729} C_VEL
LIN {X 0,Y 282.59,Z 358.723,A -85,B 0,C 180,E1 -18414.565,E2 -18414.565} C_VEL
LIN {X 0,Y 280.12,Z 372.471,A -85,B 0,C 180,E1 -18415.632,E2 -18415.632} C_VEL
LIN {X 0,Y 277.058,Z 387.091,A -85,B 0,C 180,E1 -18417.112,E2 -18417.112} C_VEL
LIN {X 0,Y 273.561,Z 400.871,A -85,B 0,C 180,E1 -18418.867,E2 -18418.867} C_VEL
LIN {X 0,Y 270.171,Z 413.102,A -85,B 0,C 180,E1 -18420.807,E2 -18420.807} C_VEL
LIN {X 0,Y 266.839,Z 424.276,A -85,B 0,C 180,E1 -18422.978,E2 -18422.978} C_VEL
LIN {X 0,Y 263.642,Z 435.128,A -85,B 0,C 180,E1 -18425.594,E2 -18425.594} C_VEL
LIN {X 0,Y 260.706,Z 444.165,A -85,B 0,C 180,E1 -18428.243,E2 -18428.243} C_VEL
LIN {X 0,Y 258.407,Z 451.671,A -85,B 0,C 180,E1 -18430.951,E2 -18430.951} C_VEL
LIN {X 0,Y 256.483,Z 458.68,A -85,B 0,C 180,E1 -18434.097,E2 -18434.097} C_VEL
LIN {X 0,Y 255.116,Z 464.195,A -85,B 0,C 180,E1 -18437.268,E2 -18437.268} C_VEL
LIN {X 0,Y 254.314,Z 468.371,A -85,B 0,C 180,E1 -18440.456,E2 -18440.456} C_VEL
LIN {X 0,Y 253.957,Z 471.302,A -85,B 0,C 180,E1 -18443.644,E2 -18443.644} C_VEL
LIN {X 0,Y 253.935,Z 473.053,A -85,B 0,C 180,E1 -18446.827,E2 -18446.827} C_VEL
LIN {X 0,Y 254.053,Z 473.654,A -85,B 0,C 180,E1 -18450,E2 -18450} C_VEL
LIN {X 0,Y 253.936,Z 473.04,A -85,B 0,C 180,E1 -18453.173,E2 -18453.173} C_VEL
LIN {X 0,Y 253.957,Z 471.273,A -85,B 0,C 180,E1 -18456.355,E2 -18456.355} C_VEL
LIN {X 0,Y 254.313,Z 468.33,A -85,B 0,C 180,E1 -18459.544,E2 -18459.544} C_VEL
LIN {X 0,Y 255.108,Z 464.146,A -85,B 0,C 180,E1 -18462.732,E2 -18462.732} C_VEL
LIN {X 0,Y 256.407,Z 458.609,A -85,B 0,C 180,E1 -18465.908,E2 -18465.908} C_VEL
LIN {X 0,Y 258.406,Z 451.576,A -85,B 0,C 180,E1 -18469.049,E2 -18469.049} C_VEL
LIN {X 0,Y 261.032,Z 442.833,A -85,B 0,C 180,E1 -18472.144,E2 -18472.144} C_VEL
LIN {X 0,Y 263.6,Z 435.006,A -85,B 0,C 180,E1 -18474.41,E2 -18474.41} C_VEL
LIN {X 0,Y 266.831,Z 424.124,A -85,B 0,C 180,E1 -18477.023,E2 -18477.023} C_VEL
LIN {X 0,Y 270.122,Z 412.927,A -85,B 0,C 180,E1 -18479.198,E2 -18479.198} C_VEL
LIN {X 0,Y 273.56,Z 400.665,A -85,B 0,C 180,E1 -18481.133,E2 -18481.133} C_VEL
LIN {X 0,Y 276.997,Z 387.096,A -85,B 0,C 180,E1 -18482.855,E2 -18482.855} C_VEL
LIN {X 0,Y 279.783,Z 373.933,A -85,B 0,C 180,E1 -18484.198,E2 -18484.198} C_VEL
LIN {X 0,Y 282.371,Z 359.438,A -85,B 0,C 180,E1 -18485.358,E2 -18485.358} C_VEL
LIN {X 0,Y 284.619,Z 344.422,A -85,B 0,C 180,E1 -18486.234,E2 -18486.234} C_VEL
LIN {X 0,Y 286.137,Z 329.889,A -85,B 0,C 180,E1 -18486.831,E2 -18486.831} C_VEL
LIN {X 0,Y 287.411,Z 305.785,A -85,B 0,C 180,E1 -18487.464,E2 -18487.464} C_VEL
LIN {X 0,Y 291.156,Z 224.896,A -85,B 0,C 180,E1 -18489.384,E2 -18489.384} C_VEL
LIN {X 0,Y 291.002,Z 222.408,A -85,B 0,C 180,E1 -18489.486,E2 -18489.486} C_VEL
LIN {X 0,Y 283.921,Z 205.977,A -85,B 0,C 180,E1 -18491.202,E2 -18491.202} C_VEL
LIN {X 0,Y 277.085,Z 192.265,A -85,B 0,C 180,E1 -18492.913,E2 -18492.913} C_VEL
LIN {X 0,Y 270.135,Z 179.667,A -85,B 0,C 180,E1 -18494.747,E2 -18494.747} C_VEL
LIN {X 0,Y 263.987,Z 169.626,A -85,B 0,C 180,E1 -18496.46,E2 -18496.46} C_VEL
LIN {X 0,Y 260.364,Z 164.068,A -85,B 0,C 180,E1 -18497.521,E2 -18497.521} C_VEL
LIN {X 0,Y 258.006,Z 160.004,A -85,B 0,C 180,E1 -18498.272,E2 -18498.272} C_VEL
LIN {X 0,Y 256.09,Z 154.203,A -85,B 0,C 180,E1 -18501.051,E2 -18501.051} C_VEL
LIN {X 0,Y 256.109,Z 154.2,A -85,B 0,C 180,E1 -18504.812,E2 -18504.812} C_VEL
LIN {X 0,Y 256.094,Z 154.208,A -85,B 0,C 180,E1 -18508.573,E2 -18508.573} C_VEL
LIN {X 0,Y 256.143,Z 154.2,A -85,B 0,C 180,E1 -18512.197,E2 -18512.197} C_VEL
LIN {X 0,Y 256.168,Z 154.196,A -85,B 0,C 180,E1 -18515.699,E2 -18515.699} C_VEL
LIN {X 0,Y 256.169,Z 154.195,A -85,B 0,C 180,E1 -18519.105,E2 -18519.105} C_VEL
LIN {X 0,Y 256.302,Z 154.175,A -85,B 0,C 180,E1 -18524.085,E2 -18524.085} C_VEL
LIN {X 0,Y 256.293,Z 154.182,A -85,B 0,C 180,E1 -18528.933,E2 -18528.933} C_VEL
LIN {X 0,Y 256.47,Z 154.152,A -85,B 0,C 180,E1 -18532.125,E2 -18532.125} C_VEL
LIN {X 0,Y 256.49,Z 154.154,A -85,B 0,C 180,E1 -18536.859,E2 -18536.859} C_VEL
LIN {X 0,Y 256.708,Z 154.134,A -85,B 0,C 180,E1 -18538.431,E2 -18538.431} C_VEL
LIN {X 0,Y 256.702,Z 154.131,A -85,B 0,C 180,E1 -18541.569,E2 -18541.569} C_VEL
LIN {X 0,Y 256.446,Z 154.162,A -85,B 0,C 180,E1 -18546.568,E2 -18546.568} C_VEL
LIN {X 0,Y 256.428,Z 154.158,A -85,B 0,C 180,E1 -18549.465,E2 -18549.465} C_VEL
LIN {X 0,Y 256.217,Z 154.19,A -85,B 0,C 180,E1 -18554.292,E2 -18554.292} C_VEL
LIN {X 0,Y 256.172,Z 154.191,A -85,B 0,C 180,E1 -18557.565,E2 -18557.565} C_VEL
LIN {X 0,Y 256.144,Z 154.195,A -85,B 0,C 180,E1 -18561.111,E2 -18561.111} C_VEL
LIN {X 0,Y 256.134,Z 154.178,A -85,B 0,C 180,E1 -18565.112,E2 -18565.112} C_VEL
LIN {X 0,Y 256.056,Z 154.215,A -85,B 0,C 180,E1 -18569.607,E2 -18569.607} C_VEL
LIN {X 0,Y 256.067,Z 154.211,A -85,B 0,C 180,E1 -18573.293,E2 -18573.293} C_VEL
LIN {X 0,Y 256.111,Z 154.2,A -85,B 0,C 180,E1 -18577.269,E2 -18577.269} C_VEL
LIN {X 0,Y 256.045,Z 154.212,A -85,B 0,C 180,E1 -18581.414,E2 -18581.414} C_VEL
LIN {X 0,Y 257.086,Z 157.136,A -85,B 0,C 180,E1 -18581.836,E2 -18581.836} C_VEL
LIN {X 0,Y 259.492,Z 159.726,A -85,B 0,C 180,E1 -18582.535,E2 -18582.535} C_VEL
LIN {X 0,Y 261.615,Z 163.054,A -85,B 0,C 180,E1 -18583.175,E2 -18583.175} C_VEL
LIN {X 0,Y 263.014,Z 164.793,A -85,B 0,C 180,E1 -18583.569,E2 -18583.569} C_VEL
LIN {X 0,Y 271.651,Z 177.341,A -85,B 0,C 180,E1 -18585.921,E2 -18585.921} C_VEL
LIN {X 0,Y 278.963,Z 188.97,A -85,B 0,C 180,E1 -18587.768,E2 -18587.768} C_VEL
LIN {X 0,Y 285.981,Z 202.652,A -85,B 0,C 180,E1 -18589.487,E2 -18589.487} C_VEL
LIN {X 0,Y 291.502,Z 214.75,A -85,B 0,C 180,E1 -18590.794,E2 -18590.794} C_VEL
LIN {X 0,Y 286.781,Z 314.959,A -85,B 0,C 180,E1 -18593.21,E2 -18593.21} C_VEL
LIN {X 0,Y 285.396,Z 330.133,A -85,B 0,C 180,E1 -18593.826,E2 -18593.826} C_VEL
LIN {X 0,Y 283.526,Z 344.877,A -85,B 0,C 180,E1 -18594.699,E2 -18594.699} C_VEL
LIN {X 0,Y 281.165,Z 359.445,A -85,B 0,C 180,E1 -18595.859,E2 -18595.859} C_VEL
LIN {X 0,Y 278.214,Z 373.808,A -85,B 0,C 180,E1 -18597.319,E2 -18597.319} C_VEL
LIN {X 0,Y 275.268,Z 386.015,A -85,B 0,C 180,E1 -18598.868,E2 -18598.868} C_VEL
LIN {X 0,Y 271.926,Z 398.428,A -85,B 0,C 180,E1 -18600.802,E2 -18600.802} C_VEL
LIN {X 0,Y 268.591,Z 409.876,A -85,B 0,C 180,E1 -18602.999,E2 -18602.999} C_VEL
LIN {X 0,Y 265.971,Z 418.451,A -85,B 0,C 180,E1 -18604.99,E2 -18604.99} C_VEL
LIN {X 0,Y 262.963,Z 427.893,A -85,B 0,C 180,E1 -18607.614,E2 -18607.614} C_VEL
LIN {X 0,Y 260.336,Z 435.751,A -85,B 0,C 180,E1 -18610.278,E2 -18610.278} C_VEL
LIN {X 0,Y 258.128,Z 443.077,A -85,B 0,C 180,E1 -18613.388,E2 -18613.388} C_VEL
LIN {X 0,Y 256.332,Z 448.889,A -85,B 0,C 180,E1 -18616.523,E2 -18616.523} C_VEL
LIN {X 0,Y 255.459,Z 452.326,A -85,B 0,C 180,E1 -18618.897,E2 -18618.897} C_VEL
LIN {X 0,Y 254.691,Z 455.802,A -85,B 0,C 180,E1 -18622.07,E2 -18622.07} C_VEL
LIN {X 0,Y 254.21,Z 458.1,A -85,B 0,C 180,E1 -18625.243,E2 -18625.243} C_VEL
LIN {X 0,Y 254.084,Z 459.269,A -85,B 0,C 180,E1 -18628.415,E2 -18628.415} C_VEL
LIN {X 0,Y 254.084,Z 459.282,A -85,B 0,C 180,E1 -18631.585,E2 -18631.585} C_VEL
LIN {X 0,Y 254.21,Z 458.166,A -85,B 0,C 180,E1 -18634.758,E2 -18634.758} C_VEL
LIN {X 0,Y 254.683,Z 455.919,A -85,B 0,C 180,E1 -18637.931,E2 -18637.931} C_VEL
LIN {X 0,Y 255.428,Z 452.489,A -85,B 0,C 180,E1 -18641.105,E2 -18641.105} C_VEL
LIN {X 0,Y 256.69,Z 447.789,A -85,B 0,C 180,E1 -18644.266,E2 -18644.266} C_VEL
LIN {X 0,Y 258.539,Z 441.692,A -85,B 0,C 180,E1 -18647.399,E2 -18647.399} C_VEL
LIN {X 0,Y 260.974,Z 434.012,A -85,B 0,C 180,E1 -18650.493,E2 -18650.493} C_VEL
LIN {X 0,Y 263.697,Z 425.817,A -85,B 0,C 180,E1 -18653.149,E2 -18653.149} C_VEL
LIN {X 0,Y 266.932,Z 415.938,A -85,B 0,C 180,E1 -18655.749,E2 -18655.749} C_VEL
LIN {X 0,Y 269.888,Z 405.813,A -85,B 0,C 180,E1 -18657.952,E2 -18657.952} C_VEL
LIN {X 0,Y 272.734,Z 395.877,A -85,B 0,C 180,E1 -18659.739,E2 -18659.739} C_VEL
LIN {X 0,Y 276.055,Z 382.932,A -85,B 0,C 180,E1 -18661.674,E2 -18661.674} C_VEL
LIN {X 0,Y 279.107,Z 370.062,A -85,B 0,C 180,E1 -18663.208,E2 -18663.208} C_VEL
LIN {X 0,Y 281.823,Z 355.589,A -85,B 0,C 180,E1 -18664.603,E2 -18664.603} C_VEL
LIN {X 0,Y 284.09,Z 341.246,A -85,B 0,C 180,E1 -18665.655,E2 -18665.655} C_VEL
LIN {X 0,Y 285.904,Z 325.95,A -85,B 0,C 180,E1 -18666.482,E2 -18666.482} C_VEL
LIN {X 0,Y 287.143,Z 311.151,A -85,B 0,C 180,E1 -18667.01,E2 -18667.01} C_VEL
LIN {X 0,Y 290.727,Z 233.238,A -85,B 0,C 180,E1 -18668.887,E2 -18668.887} C_VEL
LIN {X 0,Y 291.571,Z 214.788,A -85,B 0,C 180,E1 -18669.327,E2 -18669.327} C_VEL
LIN {X 0,Y 283.87,Z 198.167,A -85,B 0,C 180,E1 -18671.167,E2 -18671.167} C_VEL
LIN {X 0,Y 277.504,Z 186.412,A -85,B 0,C 180,E1 -18672.739,E2 -18672.739} C_VEL
LIN {X 0,Y 270.535,Z 175.603,A -85,B 0,C 180,E1 -18674.521,E2 -18674.521} C_VEL
LIN {X 0,Y 264.746,Z 167.361,A -85,B 0,C 180,E1 -18676.09,E2 -18676.09} C_VEL
LIN {X 0,Y 262.093,Z 163.544,A -85,B 0,C 180,E1 -18676.85,E2 -18676.85} C_VEL
LIN {X 0,Y 259.793,Z 160.322,A -85,B 0,C 180,E1 -18677.527,E2 -18677.527} C_VEL
LIN {X 0,Y 259.005,Z 159.131,A -85,B 0,C 180,E1 -18677.767,E2 -18677.767} C_VEL
LIN {X 0,Y 256.89,Z 156.81,A -85,B 0,C 180,E1 -18678.388,E2 -18678.388} C_VEL
LIN {X 0,Y 256.036,Z 154.201,A -85,B 0,C 180,E1 -18678.741,E2 -18678.741} C_VEL
LIN {X 0,Y 256.1,Z 154.182,A -85,B 0,C 180,E1 -18682.862,E2 -18682.862} C_VEL
LIN {X 0,Y 256.067,Z 154.199,A -85,B 0,C 180,E1 -18686.707,E2 -18686.707} C_VEL
LIN {X 0,Y 256.043,Z 154.197,A -85,B 0,C 180,E1 -18690.589,E2 -18690.589} C_VEL
LIN {X 0,Y 255.385,Z 154.298,A -85,B 0,C 180,E1 -18691.903,E2 -18691.903} C_VEL
LIN {X 0,Y 252.522,Z 154.656,A -85,B 0,C 180,E1 -18694.045,E2 -18694.045} C_VEL
LIN {X 0,Y 250.095,Z 154.958,A -85,B 0,C 180,E1 -18695.788,E2 -18695.788} C_VEL
LIN {X 0,Y 249.071,Z 155.077,A -85,B 0,C 180,E1 -18697.14,E2 -18697.14} C_VEL
LIN {X 0,Y 248.997,Z 155.084,A -85,B 0,C 180,E1 -18697.599,E2 -18697.599} C_VEL
LIN {X 0,Y 249.084,Z 155.072,A -85,B 0,C 180,E1 -18701.918,E2 -18701.918} C_VEL
LIN {X 0,Y 249.169,Z 155.065,A -85,B 0,C 180,E1 -18705.294,E2 -18705.294} C_VEL
LIN {X 0,Y 249.386,Z 155.032,A -85,B 0,C 180,E1 -18710.522,E2 -18710.522} C_VEL
LIN {X 0,Y 249.428,Z 155.04,A -85,B 0,C 180,E1 -18713.528,E2 -18713.528} C_VEL
LIN {X 0,Y 249.662,Z 155.009,A -85,B 0,C 180,E1 -18718.387,E2 -18718.387} C_VEL
LIN {X 0,Y 249.671,Z 155.006,A -85,B 0,C 180,E1 -18721.613,E2 -18721.613} C_VEL
LIN {X 0,Y 249.433,Z 155.04,A -85,B 0,C 180,E1 -18726.471,E2 -18726.471} C_VEL
LIN {X 0,Y 249.345,Z 155.04,A -85,B 0,C 180,E1 -18729.736,E2 -18729.736} C_VEL
LIN {X 0,Y 249.184,Z 155.064,A -85,B 0,C 180,E1 -18734.704,E2 -18734.704} C_VEL
LIN {X 0,Y 249.12,Z 155.069,A -85,B 0,C 180,E1 -18738.079,E2 -18738.079} C_VEL
LIN {X 0,Y 249.084,Z 155.078,A -85,B 0,C 180,E1 -18741.518,E2 -18741.518} C_VEL
LIN {X 0,Y 249.106,Z 155.076,A -85,B 0,C 180,E1 -18745.469,E2 -18745.469} C_VEL
LIN {X 0,Y 249.043,Z 155.088,A -85,B 0,C 180,E1 -18748.976,E2 -18748.976} C_VEL
LIN {X 0,Y 249.028,Z 155.088,A -85,B 0,C 180,E1 -18752.426,E2 -18752.426} C_VEL
LIN {X 0,Y 249.104,Z 155.072,A -85,B 0,C 180,E1 -18757.11,E2 -18757.11} C_VEL
LIN {X 0,Y 249.072,Z 155.083,A -85,B 0,C 180,E1 -18757.392,E2 -18757.392} C_VEL
LIN {X 0,Y 250.66,Z 160.005,A -85,B 0,C 180,E1 -18759.763,E2 -18759.763} C_VEL
LIN {X 0,Y 253.988,Z 164.948,A -85,B 0,C 180,E1 -18760.86,E2 -18760.86} C_VEL
LIN {X 0,Y 261.52,Z 176.879,A -85,B 0,C 180,E1 -18763.191,E2 -18763.191} C_VEL
LIN {X 0,Y 268.19,Z 188.301,A -85,B 0,C 180,E1 -18765.103,E2 -18765.103} C_VEL
LIN {X 0,Y 274.181,Z 199.558,A -85,B 0,C 180,E1 -18766.727,E2 -18766.727} C_VEL
LIN {X 0,Y 281.544,Z 215.043,A -85,B 0,C 180,E1 -18768.629,E2 -18768.629} C_VEL
LIN {X 0,Y 285.729,Z 225.103,A -85,B 0,C 180,E1 -18769.685,E2 -18769.685} C_VEL
LIN {X 0,Y 280.985,Z 324.067,A -85,B 0,C 180,E1 -18772.094,E2 -18772.094} C_VEL
LIN {X 0,Y 279.574,Z 339.699,A -85,B 0,C 180,E1 -18772.666,E2 -18772.666} C_VEL
LIN {X 0,Y 277.513,Z 354.726,A -85,B 0,C 180,E1 -18773.477,E2 -18773.477} C_VEL
LIN {X 0,Y 275.027,Z 368.299,A -85,B 0,C 180,E1 -18774.454,E2 -18774.454} C_VEL
LIN {X 0,Y 272.046,Z 382.763,A -85,B 0,C 180,E1 -18775.839,E2 -18775.839} C_VEL
LIN {X 0,Y 268.887,Z 395.585,A -85,B 0,C 180,E1 -18777.378,E2 -18777.378} C_VEL
LIN {X 0,Y 265.538,Z 407.599,A -85,B 0,C 180,E1 -18779.149,E2 -18779.149} C_VEL
LIN {X 0,Y 262.133,Z 418.731,A -85,B 0,C 180,E1 -18781.145,E2 -18781.145} C_VEL
LIN {X 0,Y 259.002,Z 428.916,A -85,B 0,C 180,E1 -18783.383,E2 -18783.383} C_VEL
LIN {X 0,Y 255.806,Z 439.014,A -85,B 0,C 180,E1 -18786.094,E2 -18786.094} C_VEL
LIN {X 0,Y 252.981,Z 447.342,A -85,B 0,C 180,E1 -18788.829,E2 -18788.829} C_VEL
LIN {X 0,Y 250.531,Z 455.175,A -85,B 0,C 180,E1 -18792.026,E2 -18792.026} C_VEL
LIN {X 0,Y 248.769,Z 461.413,A -85,B 0,C 180,E1 -18795.27,E2 -18795.27} C_VEL
LIN {X 0,Y 247.583,Z 466.242,A -85,B 0,C 180,E1 -18798.539,E2 -18798.539} C_VEL
LIN {X 0,Y 247.014,Z 469.788,A -85,B 0,C 180,E1 -18801.821,E2 -18801.821} C_VEL
LIN {X 0,Y 246.841,Z 472.178,A -85,B 0,C 180,E1 -18805.21,E2 -18805.21} C_VEL
LIN {X 0,Y 246.919,Z 473.3,A -85,B 0,C 180,E1 -18808.369,E2 -18808.369} C_VEL
LIN {X 0,Y 246.982,Z 473.456,A -85,B 0,C 180,E1 -18810,E2 -18810} C_VEL
LIN {X 0,Y 246.838,Z 472.841,A -85,B 0,C 180,E1 -18813.264,E2 -18813.264} C_VEL
LIN {X 0,Y 246.872,Z 471.073,A -85,B 0,C 180,E1 -18816.539,E2 -18816.539} C_VEL
LIN {X 0,Y 247.268,Z 468.13,A -85,B 0,C 180,E1 -18819.819,E2 -18819.819} C_VEL
LIN {X 0,Y 248.14,Z 463.945,A -85,B 0,C 180,E1 -18823.096,E2 -18823.096} C_VEL
LIN {X 0,Y 249.5,Z 458.406,A -85,B 0,C 180,E1 -18826.361,E2 -18826.361} C_VEL
LIN {X 0,Y 251.647,Z 451.374,A -85,B 0,C 180,E1 -18829.581,E2 -18829.581} C_VEL
LIN {X 0,Y 254.432,Z 442.631,A -85,B 0,C 180,E1 -18832.75,E2 -18832.75} C_VEL
LIN {X 0,Y 257.056,Z 434.803,A -85,B 0,C 180,E1 -18835.073,E2 -18835.073} C_VEL
LIN {X 0,Y 260.471,Z 423.921,A -85,B 0,C 180,E1 -18837.739,E2 -18837.739} C_VEL
LIN {X 0,Y 264.209,Z 411.694,A -85,B 0,C 180,E1 -18840.138,E2 -18840.138} C_VEL
LIN {X 0,Y 267.816,Z 399.232,A -85,B 0,C 180,E1 -18842.1,E2 -18842.1} C_VEL
LIN {X 0,Y 271.312,Z 385.686,A -85,B 0,C 180,E1 -18843.81,E2 -18843.81} C_VEL
LIN {X 0,Y 274.298,Z 371.892,A -85,B 0,C 180,E1 -18845.204,E2 -18845.204} C_VEL
LIN {X 0,Y 276.816,Z 358.096,A -85,B 0,C 180,E1 -18846.29,E2 -18846.29} C_VEL
LIN {X 0,Y 279.155,Z 342.653,A -85,B 0,C 180,E1 -18847.173,E2 -18847.173} C_VEL
LIN {X 0,Y 280.682,Z 327.361,A -85,B 0,C 180,E1 -18847.783,E2 -18847.783} C_VEL
LIN {X 0,Y 284.4,Z 251.51,A -85,B 0,C 180,E1 -18849.644,E2 -18849.644} C_VEL
LIN {X 0,Y 285.62,Z 225.043,A -85,B 0,C 180,E1 -18850.29,E2 -18850.29} C_VEL
LIN {X 0,Y 278.787,Z 208.994,A -85,B 0,C 180,E1 -18852.023,E2 -18852.023} C_VEL
LIN {X 0,Y 271.861,Z 195.157,A -85,B 0,C 180,E1 -18853.834,E2 -18853.834} C_VEL
LIN {X 0,Y 266.018,Z 184.499,A -85,B 0,C 180,E1 -18855.444,E2 -18855.444} C_VEL
LIN {X 0,Y 259.677,Z 173.986,A -85,B 0,C 180,E1 -18857.289,E2 -18857.289} C_VEL
LIN {X 0,Y 256.167,Z 168.539,A -85,B 0,C 180,E1 -18858.363,E2 -18858.363} C_VEL
LIN {X 0,Y 253.694,Z 164.572,A -85,B 0,C 180,E1 -18859.158,E2 -18859.158} C_VEL
LIN {X 0,Y 250.468,Z 159.624,A -85,B 0,C 180,E1 -18860.266,E2 -18860.266} C_VEL
LIN {X 0,Y 249.077,Z 155.08,A -85,B 0,C 180,E1 -18862.613,E2 -18862.613} C_VEL
LIN {X 0,Y 249.057,Z 155.084,A -85,B 0,C 180,E1 -18865.642,E2 -18865.642} C_VEL
LIN {X 0,Y 249.053,Z 155.078,A -85,B 0,C 180,E1 -18869.474,E2 -18869.474} C_VEL
LIN {X 0,Y 249.075,Z 155.076,A -85,B 0,C 180,E1 -18873.163,E2 -18873.163} C_VEL
LIN {X 0,Y 249.081,Z 155.076,A -85,B 0,C 180,E1 -18876.733,E2 -18876.733} C_VEL
LIN {X 0,Y 249.112,Z 155.07,A -85,B 0,C 180,E1 -18880.212,E2 -18880.212} C_VEL
LIN {X 0,Y 249.244,Z 155.053,A -85,B 0,C 180,E1 -18883.622,E2 -18883.622} C_VEL
LIN {X 0,Y 249.237,Z 155.058,A -85,B 0,C 180,E1 -18888.616,E2 -18888.616} C_VEL
